  MoveL 631 to (-33.29, -26.54, 35) mm, rotated rx 180 ry 0 rz -180 deg; joints [31.763, 57.392, 24.529, -147.981, 83.138, -184.273]
  Call Extruder(6882.338)
  MoveL 632 to (-26.54, -33.28, 35) mm, rotated rx 180 ry 0 rz -180 deg; joints [30.206, 57.574, 23.981, -149.522, 82.708, -184.272]
  Call Extruder(6897.234)
  MoveL 633 to (-18.47, -38.36, 35) mm, rotated rx 180 ry 0 rz 180 deg; joints [28.808, 57.937, 22.898, -150.881, 81.977, -184.445]
  Call Extruder(6912.129)
  MoveL 634 to (-9.47, -41.5, 35) mm, rotated rx 180 ry 0 rz 180 deg; joints [27.654, 58.472, 21.339, -151.97, 80.985, -184.769]
  Call Extruder(6927.025)
  MoveL 635 to (0, -42.57, 35) mm, rotated rx 180 ry 0 rz 180 deg; joints [26.805, 59.159, 19.387, -152.729, 79.791, -185.221]
  Call Extruder(6928.241)
  MoveL 636 to (0.77, -42.49, 35) mm, rotated rx -180 ry 0 rz 180 deg; joints [26.762, 59.224, 19.206, -152.762, 79.683, -185.267]
  Call Extruder(6941.921)
  MoveL 637 to (9.47, -41.5, 35) mm, rotated rx 180 ry 0 rz -180 deg; joints [26.29, 59.972, 17.142, -153.125, 78.466, -185.786]
  Call Extruder(6956.817)
  MoveL 638 to (18.47, -38.36, 35) mm, rotated rx -180 ry 0 rz -180 deg; joints [26.114, 60.875, 14.715, -153.155, 77.088, -186.452]
  Call Extruder(6971.713)
  MoveL 639 to (26.54, -33.28, 35) mm, rotated rx -180 ry 0 rz -180 deg; joints [26.262, 61.827, 12.225, -152.835, 75.735, -187.206]
  Call Extruder(6986.609)
  MoveL 640 to (33.28, -26.54, 35) mm, rotated rx 180 ry 0 rz 180 deg; joints [26.703, 62.779, 9.793, -152.201, 74.481, -188.03]
  Call Extruder(7001.504)
  MoveL 641 to (38.36, -18.47, 35) mm, rotated rx 180 ry 0 rz -180 deg; joints [27.4, 63.681, 7.536, -151.299, 73.389, -188.896]
  Call Extruder(7016.400)
  MoveL 642 to (41.5, -9.47, 35) mm, rotated rx -180 ry 0 rz -180 deg; joints [28.309, 64.481, 5.567, -150.186, 72.517, -189.768]
  Call Extruder(7031.296)
  MoveL 643 to (42.57, 0, 35) mm, rotated rx -180 ry 0 rz 180 deg; joints [29.382, 65.132, 3.985, -148.925, 71.904, -190.602]
  Call Extruder(7046.192)
  MoveL 644 to (41.51, 9.47, 35) mm, rotated rx -180 ry 0 rz -180 deg; joints [30.575, 65.593, 2.875, -147.579, 71.579, -191.348]
  Call Extruder(7061.087)
  MoveL 645 to (38.36, 18.47, 35) mm, rotated rx -180 ry 0 rz -180 deg; joints [31.839, 65.836, 2.295, -146.213, 71.552, -191.955]
  Call Extruder(7075.983)
  MoveL 646 to (33.28, 26.54, 35) mm, rotated rx 180 ry 0 rz -180 deg; joints [33.128, 65.843, 2.278, -144.884, 71.816, -192.378]
  Call Extruder(7090.879)
  MoveL 647 to (26.54, 33.29, 35) mm, rotated rx 180 ry 0 rz -180 deg; joints [34.394, 65.614, 2.825, -143.644, 72.348, -192.583]
  Call Extruder(7105.775)
  MoveL 648 to (18.47, 38.36, 35) mm, rotated rx 180 ry 0 rz -180 deg; joints [35.592, 65.165, 3.906, -142.537, 73.113, -192.549]
  Call Extruder(7120.671)
  MoveL 649 to (9.47, 41.5, 35) mm, rotated rx 180 ry 0 rz 180 deg; joints [36.675, 64.524, 5.462, -141.601, 74.068, -192.274]
  Call Extruder(7135.566)
  MoveL 650 to (0, 42.57, 35) mm, rotated rx 180 ry 0 rz 180 deg; joints [37.594, 63.731, 7.411, -140.868, 75.161, -191.77]
  Call Extruder(7150.462)
  MoveL 651 to (-9.47, 41.5, 35) mm, rotated rx 180 ry 0 rz 180 deg; joints [38.304, 62.834, 9.654, -140.366, 76.342, -191.066]
  Call Extruder(7165.358)
  MoveL 652 to (-18.47, 38.36, 35) mm, rotated rx 180 ry 0 rz -180 deg; joints [38.762, 61.883, 12.079, -140.123, 77.56, -190.202]
  Call Extruder(7180.254)
  MoveL 653 to (-26.54, 33.29, 35) mm, rotated rx 180 ry 0 rz -180 deg; joints [38.928, 60.93, 14.569, -140.162, 78.768, -189.23]
  Call Extruder(7195.150)
  MoveL 654 to (-33.29, 26.54, 35) mm, rotated rx -180 ry 0 rz 180 deg; joints [38.772, 60.023, 17.003, -140.502, 79.919, -188.21]
  Call Extruder(7210.046)
  MoveL 655 to (-38.36, 18.47, 35) mm, rotated rx -180 ry 0 rz 180 deg; joints [38.277, 59.204, 19.262, -141.153, 80.969, -187.205]
  Call Extruder(7224.941)
  MoveL 656 to (-41.51, 9.47, 35) mm, rotated rx 180 ry 0 rz 180 deg; joints [37.447, 58.508, 21.234, -142.107, 81.872, -186.279]
  Call Extruder(7239.837)
  MoveL 657 to (-42.57, 0, 35) mm, rotated rx 180 ry 0 rz -180 deg; joints [36.31, 57.964, 22.819, -143.334, 82.584, -185.489]
  Call Extruder(7247.391)
  MoveL 658 to (-42.03, -4.8, 35) mm, rotated rx 180 ry 0 rz 180 deg; joints [35.612, 57.771, 23.391, -144.064, 82.824, -185.174]
  Set speed (130.0 mm/s)
  MoveL 659 to (-54.1, -7.67, 35) mm, rotated rx 180 ry 0 rz -180 deg; joints [36.421, 56.883, 26.099, -143.373, 84.357, -184.181]
  Call Extruder(7251.464)
  Set speed (30.0 mm/s)
  MoveL 660 to (-53.59, -12.23, 35) mm, rotated rx 180 ry 0 rz -180 deg; joints [35.732, 56.714, 26.627, -144.084, 84.599, -183.9]
  Call Extruder(7262.394)
  MoveL 661 to (-49.53, -23.85, 35) mm, rotated rx 180 ry 0 rz -180 deg; joints [33.663, 56.476, 27.386, -146.185, 84.894, -183.411]
  Call Extruder(7273.324)
  MoveL 662 to (-42.98, -34.27, 35) mm, rotated rx -180 ry 0 rz 180 deg; joints [31.506, 56.469, 27.408, -148.348, 84.782, -183.209]
  Call Extruder(7284.255)
  MoveL 663 to (-34.27, -42.98, 35) mm, rotated rx 180 ry 0 rz 180 deg; joints [29.427, 56.694, 26.692, -150.409, 84.242, -183.261]
  Call Extruder(7295.185)
  MoveL 664 to (-23.85, -49.52, 35) mm, rotated rx 180 ry 0 rz 180 deg; joints [27.581, 57.146, 25.28, -152.213, 83.292, -183.522]
  Call Extruder(7306.115)
  MoveL 665 to (-12.23, -53.59, 35) mm, rotated rx 180 ry 0 rz 180 deg; joints [26.087, 57.817, 23.254, -153.636, 81.987, -183.952]
  Call Extruder(7317.045)
  MoveL 666 to (0, -54.97, 35) mm, rotated rx 180 ry 0 rz -180 deg; joints [25.019, 58.686, 20.723, -154.602, 80.413, -184.521]
  Call Extruder(7318.968)
  MoveL 667 to (2.15, -54.73, 35) mm, rotated rx 180 ry 0 rz -180 deg; joints [24.908, 58.864, 20.219, -154.69, 80.109, -184.644]
  Call Extruder(7327.975)
  MoveL 668 to (12.23, -53.59, 35) mm, rotated rx 180 ry 0 rz 180 deg; joints [24.406, 59.724, 17.819, -155.077, 78.672, -185.215]
  Call Extruder(7338.905)
  MoveL 669 to (23.85, -49.53, 35) mm, rotated rx -180 ry 0 rz 180 deg; joints [24.239, 60.887, 14.685, -155.066, 76.867, -186.03]
  Call Extruder(7349.836)
  MoveL 670 to (34.27, -42.98, 35) mm, rotated rx 180 ry 0 rz 180 deg; joints [24.487, 62.12, 11.47, -154.602, 75.102, -186.96]
  Call Extruder(7360.766)
  MoveL 671 to (42.98, -34.27, 35) mm, rotated rx 180 ry 0 rz 180 deg; joints [25.101, 63.363, 8.326, -153.736, 73.471, -187.991]
  Call Extruder(7371.696)
  MoveL 672 to (49.52, -23.85, 35) mm, rotated rx 180 ry 0 rz 180 deg; joints [26.025, 64.548, 5.404, -152.536, 72.058, -189.097]
  Call Extruder(7382.626)
  MoveL 673 to (53.59, -12.23, 35) mm, rotated rx -180 ry 0 rz -180 deg; joints [27.2, 65.605, 2.847, -151.077, 70.933, -190.232]
  Call Extruder(7393.557)
  MoveL 674 to (54.97, 0, 35) mm, rotated rx 180 ry 0 rz -180 deg; joints [28.57, 66.47, 0.786, -149.44, 70.152, -191.336]
  Call Extruder(7404.487)
  MoveL 675 to (53.59, 12.23, 35) mm, rotated rx 180 ry 0 rz 180 deg; joints [30.077, 67.087, -0.665, -147.712, 69.749, -192.338]
  Call Extruder(7415.417)
  MoveL 676 to (49.52, 23.85, 35) mm, rotated rx -180 ry 0 rz -180 deg; joints [31.665, 67.411, -1.424, -145.972, 69.735, -193.163]
  Call Extruder(7426.347)
  MoveL 677 to (42.98, 34.27, 35) mm, rotated rx 180 ry 0 rz -180 deg; joints [33.282, 67.42, -1.445, -144.295, 70.101, -193.745]
  Call Extruder(7437.277)
  MoveL 678 to (34.27, 42.98, 35) mm, rotated rx 180 ry 0 rz -180 deg; joints [34.874, 67.114, -0.729, -142.742, 70.813, -194.035]
  Call Extruder(7448.208)
  MoveL 679 to (23.85, 49.53, 35) mm, rotated rx 180 ry 0 rz -180 deg; joints [36.387, 66.514, 0.683, -141.362, 71.82, -194.004]
  Call Extruder(7459.138)
  MoveL 680 to (12.23, 53.59, 35) mm, rotated rx -180 ry 0 rz -180 deg; joints [37.766, 65.662, 2.71, -140.192, 73.06, -193.649]
  Call Extruder(7470.068)
  MoveL 681 to (0, 54.97, 35) mm, rotated rx -180 ry 0 rz -180 deg; joints [38.954, 64.614, 5.242, -139.267, 74.466, -192.987]
  Call Extruder(7480.998)
  MoveL 682 to (-12.23, 53.59, 35) mm, rotated rx 180 ry 0 rz -180 deg; joints [39.895, 63.435, 8.147, -138.616, 75.972, -192.056]
  Call Extruder(7491.928)
  MoveL 683 to (-23.85, 49.52, 35) mm, rotated rx -180 ry 0 rz 180 deg; joints [40.528, 62.194, 11.282, -138.274, 77.515, -190.912]
  Call Extruder(7502.859)
  MoveL 684 to (-34.27, 42.98, 35) mm, rotated rx 180 ry 0 rz 180 deg; joints [40.799, 60.958, 14.496, -138.275, 79.04, -189.622]
  Call Extruder(7513.789)
  MoveL 685 to (-42.98, 34.27, 35) mm, rotated rx 180 ry 0 rz 180 deg; joints [40.659, 59.789, 17.64, -138.653, 80.496, -188.267]
  Call Extruder(7524.719)
  MoveL 686 to (-49.53, 23.85, 35) mm, rotated rx -180 ry 0 rz -180 deg; joints [40.072, 58.743, 20.561, -139.432, 81.835, -186.932]
  Call Extruder(7535.649)
  MoveL 687 to (-53.59, 12.23, 35) mm, rotated rx 180 ry 0 rz 180 deg; joints [39.031, 57.863, 23.118, -140.62, 83.005, -185.708]
  Call Extruder(7546.579)
  MoveL 688 to (-54.97, 0, 35) mm, rotated rx 180 ry 0 rz 180 deg; joints [37.56, 57.18, 25.177, -142.193, 83.948, -184.676]
  Call Extruder(7552.105)
  MoveL 689 to (-54.27, -6.18, 35) mm, rotated rx 180 ry 0 rz -180 deg; joints [36.644, 56.939, 25.923, -143.142, 84.278, -184.275]
  Set speed (130.0 mm/s)
  MoveL 690 to (-49.9, -9.51, 35) mm, rotated rx 180 ry 0 rz 180 deg; joints [35.741, 57.057, 25.556, -144.032, 84.01, -184.331]
  MoveL 691 to (2.97, -12.99, 35) mm, rotated rx 180 ry 0 rz 180 deg; joints [30.614, 60.72, 15.128, -148.606, 77.853, -187.317]
  Call Extruder(7556.769)
  Set speed (80.0 mm/s)
  MoveL 692 to (5.78, -12.01, 35) mm, rotated rx 180 ry 0 rz 180 deg; joints [30.526, 61.006, 14.369, -148.642, 77.438, -187.55]
  Call Extruder(7561.432)
  MoveL 693 to (8.31, -10.42, 35) mm, rotated rx -180 ry 0 rz 180 deg; joints [30.538, 61.302, 13.59, -148.572, 77.027, -187.811]
  Call Extruder(7566.096)
  MoveL 694 to (10.42, -8.31, 35) mm, rotated rx 180 ry 0 rz 180 deg; joints [30.649, 61.594, 12.829, -148.402, 76.643, -188.088]
  Call Extruder(7570.760)
  MoveL 695 to (12.01, -5.78, 35) mm, rotated rx 180 ry 0 rz 180 deg; joints [30.85, 61.866, 12.124, -148.143, 76.304, -188.37]
  Call Extruder(7575.424)
  MoveL 696 to (12.99, -2.97, 35) mm, rotated rx 180 ry 0 rz -180 deg; joints [31.131, 62.104, 11.511, -147.808, 76.027, -188.643]
  Call Extruder(7580.087)
  MoveL 697 to (13.33, 0, 35) mm, rotated rx -180 ry 0 rz 180 deg; joints [31.476, 62.296, 11.021, -147.416, 75.828, -188.894]
  Call Extruder(7584.751)
  MoveL 698 to (12.99, 2.97, 35) mm, rotated rx -180 ry 0 rz -180 deg; joints [31.869, 62.43, 10.678, -146.987, 75.714, -189.109]
  Call Extruder(7589.415)
  MoveL 699 to (12.01, 5.78, 35) mm, rotated rx 180 ry 0 rz -180 deg; joints [32.292, 62.5, 10.5, -146.541, 75.691, -189.276]
  Call Extruder(7594.079)
  MoveL 700 to (10.42, 8.31, 35) mm, rotated rx 180 ry 0 rz 180 deg; joints [32.725, 62.502, 10.494, -146.1, 75.758, -189.387]
  Call Extruder(7598.743)
  MoveL 701 to (8.31, 10.42, 35) mm, rotated rx 180 ry 0 rz 180 deg; joints [33.149, 62.436, 10.663, -145.683, 75.912, -189.433]
  Call Extruder(7603.406)
  MoveL 702 to (5.78, 12.01, 35) mm, rotated rx 180 ry 0 rz -180 deg; joints [33.544, 62.305, 10.997, -145.309, 76.144, -189.412]
  Call Extruder(7608.070)
  MoveL 703 to (2.97, 13, 35) mm, rotated rx 180 ry 0 rz 180 deg; joints [33.893, 62.117, 11.479, -144.996, 76.442, -189.323]
  Call Extruder(7612.734)
  MoveL 704 to (0, 13.33, 35) mm, rotated rx 180 ry 0 rz 180 deg; joints [34.177, 61.881, 12.085, -144.758, 76.791, -189.171]
  Call Extruder(7617.398)
  MoveL 705 to (-2.97, 13, 35) mm, rotated rx 180 ry 0 rz -180 deg; joints [34.384, 61.611, 12.785, -144.607, 77.174, -188.963]
  Call Extruder(7622.062)
  MoveL 706 to (-5.78, 12.01, 35) mm, rotated rx 180 ry 0 rz -180 deg; joints [34.5, 61.32, 13.544, -144.55, 77.573, -188.711]
  Call Extruder(7626.725)
  MoveL 707 to (-8.31, 10.42, 35) mm, rotated rx -180 ry 0 rz 180 deg; joints [34.518, 61.023, 14.324, -144.592, 77.97, -188.428]
  Call Extruder(7631.389)
  MoveL 708 to (-10.42, 8.31, 35) mm, rotated rx 180 ry 0 rz 180 deg; joints [34.436, 60.736, 15.085, -144.733, 78.344, -188.131]
  Call Extruder(7636.053)
  MoveL 709 to (-12.01, 5.78, 35) mm, rotated rx 180 ry 0 rz -180 deg; joints [34.254, 60.472, 15.79, -144.968, 78.68, -187.835]
  Call Extruder(7640.717)
  MoveL 710 to (-13, 2.97, 35) mm, rotated rx -180 ry 0 rz -180 deg; joints [33.981, 60.244, 16.404, -145.287, 78.96, -187.557]
  Call Extruder(7645.380)
  MoveL 711 to (-13.33, 0, 35) mm, rotated rx 180 ry 0 rz -180 deg; joints [33.63, 60.063, 16.894, -145.676, 79.169, -187.311]
  Call Extruder(7650.044)
  MoveL 712 to (-13, -2.97, 35) mm, rotated rx 180 ry 0 rz 180 deg; joints [33.218, 59.936, 17.238, -146.116, 79.297, -187.109]
  Call Extruder(7654.708)
  MoveL 713 to (-12.01, -5.78, 35) mm, rotated rx 180 ry 0 rz -180 deg; joints [32.767, 59.871, 17.417, -146.583, 79.337, -186.961]
  Call Extruder(7659.372)
  MoveL 714 to (-10.42, -8.31, 35) mm, rotated rx 180 ry 0 rz -180 deg; joints [32.302, 59.869, 17.422, -147.052, 79.283, -186.872]
  Call Extruder(7664.036)
  MoveL 715 to (-8.31, -10.42, 35) mm, rotated rx 180 ry 0 rz 180 deg; joints [31.85, 59.931, 17.253, -147.498, 79.139, -186.845]
  Call Extruder(7668.699)
  MoveL 716 to (-5.78, -12.01, 35) mm, rotated rx -180 ry 0 rz -180 deg; joints [31.435, 60.054, 16.919, -147.896, 78.911, -186.881]
  Call Extruder(7673.363)
  MoveL 717 to (-2.97, -12.99, 35) mm, rotated rx 180 ry 0 rz -180 deg; joints [31.079, 60.232, 16.436, -148.224, 78.61, -186.975]
  Call Extruder(7678.027)
  MoveL 718 to (0, -13.33, 35) mm, rotated rx 180 ry 0 rz 180 deg; joints [30.801, 60.457, 15.829, -148.465, 78.251, -187.123]
  Call Extruder(7682.691)
  MoveL 719 to (2.97, -12.99, 35) mm, rotated rx 180 ry 0 rz 180 deg; joints [30.614, 60.72, 15.128, -148.606, 77.853, -187.317]
  Set speed (130.0 mm/s)
  MoveL 720 to (2.97, -12.99, 40) mm, rotated rx 180 ry 0 rz 180 deg; joints [30.614, 59.777, 15.612, -148.554, 77.462, -187.562]
  MoveL 721 to (-26.25, -4.54, 40) mm, rotated rx 180 ry 0 rz 180 deg; joints [34.172, 57.891, 20.698, -145.294, 80.579, -186.468]
  Call Extruder(7684.924)
  Set speed (60.0 mm/s)
  MoveL 722 to (-26.09, -5.96, 40) mm, rotated rx 180 ry 0 rz -180 deg; joints [33.969, 57.832, 20.861, -145.509, 80.642, -186.374]
  Call Extruder(7694.288)
  MoveL 723 to (-24.12, -11.61, 40) mm, rotated rx -180 ry 0 rz -180 deg; joints [33.033, 57.703, 21.223, -146.473, 80.733, -186.09]
  Call Extruder(7703.653)
  MoveL 724 to (-20.93, -16.69, 40) mm, rotated rx 180 ry 0 rz 180 deg; joints [32.066, 57.699, 21.234, -147.448, 80.638, -185.928]
  Call Extruder(7713.018)
  MoveL 725 to (-16.69, -20.93, 40) mm, rotated rx 180 ry 0 rz -180 deg; joints [31.126, 57.821, 20.892, -148.376, 80.355, -185.89]
  Call Extruder(7722.383)
  MoveL 726 to (-11.61, -24.11, 40) mm, rotated rx 180 ry 0 rz -180 deg; joints [30.272, 58.064, 20.217, -149.2, 79.897, -185.97]
  Call Extruder(7731.748)
  MoveL 727 to (-5.96, -26.09, 40) mm, rotated rx 180 ry 0 rz -180 deg; joints [29.552, 58.419, 19.242, -149.87, 79.287, -186.158]
  Call Extruder(7741.113)
  MoveL 728 to (0, -26.77, 40) mm, rotated rx 180 ry 0 rz 180 deg; joints [29.003, 58.87, 18.019, -150.351, 78.558, -186.443]
  Call Extruder(7745.379)
  MoveL 729 to (2.71, -26.46, 40) mm, rotated rx -180 ry 0 rz 180 deg; joints [28.841, 59.109, 17.38, -150.474, 78.191, -186.612]
  Call Extruder(7750.478)
  MoveL 730 to (5.96, -26.09, 40) mm, rotated rx -180 ry 0 rz -180 deg; joints [28.65, 59.398, 16.61, -150.618, 77.75, -186.813]
  Call Extruder(7759.843)
  MoveL 731 to (11.61, -24.11, 40) mm, rotated rx -180 ry 0 rz -180 deg; joints [28.503, 59.979, 15.084, -150.664, 76.908, -187.255]
  Call Extruder(7769.208)
  MoveL 732 to (16.69, -20.93, 40) mm, rotated rx 180 ry 0 rz 180 deg; joints [28.559, 60.584, 13.519, -150.493, 76.079, -187.754]
  Call Extruder(7778.573)
  MoveL 733 to (20.93, -16.69, 40) mm, rotated rx 180 ry 0 rz -180 deg; joints [28.808, 61.183, 11.99, -150.121, 75.307, -188.291]
  Call Extruder(7787.938)
  MoveL 734 to (24.12, -11.61, 40) mm, rotated rx -180 ry 0 rz 180 deg; joints [29.229, 61.746, 10.575, -149.575, 74.632, -188.846]
  Call Extruder(7797.303)
  MoveL 735 to (26.09, -5.96, 40) mm, rotated rx -180 ry 0 rz 180 deg; joints [29.796, 62.241, 9.343, -148.888, 74.089, -189.395]
  Call Extruder(7806.668)
  MoveL 736 to (26.77, 0, 40) mm, rotated rx 180 ry 0 rz 180 deg; joints [30.482, 62.641, 8.356, -148.096, 73.703, -189.909]
  Call Extruder(7816.033)
  MoveL 737 to (26.09, 5.96, 40) mm, rotated rx 180 ry 0 rz -180 deg; joints [31.252, 62.923, 7.666, -147.241, 73.493, -190.36]
  Call Extruder(7825.398)
  MoveL 738 to (24.11, 11.61, 40) mm, rotated rx -180 ry 0 rz -180 deg; joints [32.076, 63.07, 7.305, -146.362, 73.466, -190.722]
  Call Extruder(7834.763)
  MoveL 739 to (20.93, 16.69, 40) mm, rotated rx -180 ry 0 rz 180 deg; joints [32.917, 63.074, 7.295, -145.499, 73.619, -190.97]
  Call Extruder(7844.128)
  MoveL 740 to (16.69, 20.93, 40) mm, rotated rx 180 ry 0 rz 180 deg; joints [33.742, 62.935, 7.635, -144.689, 73.942, -191.086]
  Call Extruder(7853.493)
  MoveL 741 to (11.61, 24.12, 40) mm, rotated rx 180 ry 0 rz -180 deg; joints [34.517, 62.661, 8.307, -143.964, 74.414, -191.06]
  Call Extruder(7862.858)
  MoveL 742 to (5.96, 26.09, 40) mm, rotated rx 180 ry 0 rz 180 deg; joints [35.208, 62.267, 9.278, -143.354, 75.01, -190.891]
  Call Extruder(7872.223)
  MoveL 743 to (0, 26.77, 40) mm, rotated rx 180 ry 0 rz -180 deg; joints [35.784, 61.777, 10.497, -142.884, 75.701, -190.587]
  Call Extruder(7881.588)
  MoveL 744 to (-5.96, 26.09, 40) mm, rotated rx 180 ry 0 rz -180 deg; joints [36.214, 61.218, 11.903, -142.576, 76.452, -190.163]
  Call Extruder(7890.953)
  MoveL 745 to (-11.61, 24.12, 40) mm, rotated rx 180 ry 0 rz 180 deg; joints [36.473, 60.62, 13.427, -142.445, 77.231, -189.644]
  Call Extruder(7900.318)
  MoveL 746 to (-16.69, 20.93, 40) mm, rotated rx 180 ry 0 rz 180 deg; joints [36.542, 60.014, 14.993, -142.504, 78.004, -189.06]
  Call Extruder(7909.683)
  MoveL 747 to (-20.93, 16.69, 40) mm, rotated rx 180 ry 0 rz -180 deg; joints [36.407, 59.431, 16.522, -142.759, 78.736, -188.446]
  Call Extruder(7919.048)
  MoveL 748 to (-24.12, 11.61, 40) mm, rotated rx -180 ry 0 rz -180 deg; joints [36.065, 58.899, 17.941, -143.206, 79.395, -187.837]
  Call Extruder(7928.413)
  MoveL 749 to (-26.09, 5.96, 40) mm, rotated rx -180 ry 0 rz 180 deg; joints [35.528, 58.443, 19.177, -143.832, 79.951, -187.269]
  Call Extruder(7937.778)
  MoveL 750 to (-26.77, 0, 40) mm, rotated rx -180 ry 0 rz -180 deg; joints [34.817, 58.082, 20.167, -144.612, 80.375, -186.773]
  Call Extruder(7942.567)
  MoveL 751 to (-26.42, -3.05, 40) mm, rotated rx 180 ry 0 rz -180 deg; joints [34.385, 57.953, 20.525, -145.069, 80.512, -186.567]
  Set speed (130.0 mm/s)
  MoveL 752 to (-41.86, -6.29, 40) mm, rotated rx 180 ry 0 rz 180 deg; joints [35.393, 56.711, 24.057, -144.253, 82.485, -185.378]
  Call Extruder(7947.564)
  Set speed (60.0 mm/s)
  MoveL 753 to (-41.51, -9.47, 40) mm, rotated rx 180 ry 0 rz 180 deg; joints [34.924, 56.586, 24.424, -144.743, 82.639, -185.175]
  Call Extruder(7962.460)
  MoveL 754 to (-38.36, -18.47, 40) mm, rotated rx 180 ry 0 rz 180 deg; joints [33.373, 56.389, 25.006, -146.328, 82.822, -184.759]
  Call Extruder(7977.356)
  MoveL 755 to (-33.29, -26.54, 40) mm, rotated rx 180 ry 0 rz 180 deg; joints [31.763, 56.383, 25.023, -147.947, 82.701, -184.549]
  Call Extruder(7992.252)
  MoveL 756 to (-26.54, -33.28, 40) mm, rotated rx 180 ry 0 rz 180 deg; joints [30.206, 56.569, 24.474, -149.487, 82.267, -184.534]
  Call Extruder(8007.148)
  MoveL 757 to (-18.47, -38.36, 40) mm, rotated rx 180 ry 0 rz 180 deg; joints [28.808, 56.941, 23.389, -150.845, 81.536, -184.694]
  Call Extruder(8022.043)
  MoveL 758 to (-9.47, -41.51, 40) mm, rotated rx 180 ry 0 rz 180 deg; joints [27.654, 57.488, 21.827, -151.932, 80.548, -185.005]
  Call Extruder(8036.939)
  MoveL 759 to (0, -42.57, 40) mm, rotated rx 180 ry 0 rz 180 deg; joints [26.805, 58.189, 19.873, -152.688, 79.361, -185.446]
  Call Extruder(8043.970)
  MoveL 760 to (4.47, -42.07, 40) mm, rotated rx 180 ry 0 rz 180 deg; joints [26.559, 58.574, 18.819, -152.878, 78.742, -185.71]
  Call Extruder(8051.835)
  MoveL 761 to (9.47, -41.5, 40) mm, rotated rx 180 ry 0 rz -180 deg; joints [26.29, 59.017, 17.626, -153.081, 78.046, -186.004]
  Call Extruder(8066.731)
  MoveL 762 to (18.47, -38.36, 40) mm, rotated rx 180 ry 0 rz 180 deg; joints [26.114, 59.935, 15.198, -153.107, 76.681, -186.664]
  Call Extruder(8081.626)
  MoveL 763 to (26.54, -33.28, 40) mm, rotated rx 180 ry 0 rz 180 deg; joints [26.262, 60.901, 12.708, -152.783, 75.341, -187.415]
  Call Extruder(8096.522)
  MoveL 764 to (33.28, -26.54, 40) mm, rotated rx 180 ry 0 rz 180 deg; joints [26.703, 61.865, 10.277, -152.144, 74.1, -188.238]
  Call Extruder(8111.418)
  MoveL 765 to (38.36, -18.47, 40) mm, rotated rx 180 ry 0 rz 180 deg; joints [27.4, 62.777, 8.021, -151.238, 73.023, -189.105]
  Call Extruder(8126.314)
  MoveL 766 to (41.51, -9.47, 40) mm, rotated rx -180 ry 0 rz 180 deg; joints [28.309, 63.586, 6.054, -150.121, 72.163, -189.981]
  Call Extruder(8141.210)
  MoveL 767 to (42.57, 0, 40) mm, rotated rx 180 ry 0 rz 180 deg; joints [29.382, 64.243, 4.474, -148.856, 71.562, -190.82]
  Call Extruder(8156.106)
  MoveL 768 to (41.5, 9.47, 40) mm, rotated rx 180 ry 0 rz 180 deg; joints [30.575, 64.709, 3.365, -147.508, 71.247, -191.571]
  Call Extruder(8171.001)
  MoveL 769 to (38.36, 18.47, 40) mm, rotated rx -180 ry 0 rz 180 deg; joints [31.839, 64.953, 2.786, -146.139, 71.227, -192.185]
  Call Extruder(8185.897)
  MoveL 770 to (33.28, 26.54, 40) mm, rotated rx 180 ry 0 rz -180 deg; joints [33.128, 64.96, 2.77, -144.809, 71.496, -192.615]
  Call Extruder(8200.793)
  MoveL 771 to (26.54, 33.29, 40) mm, rotated rx 180 ry 0 rz -180 deg; joints [34.394, 64.729, 3.316, -143.569, 72.031, -192.828]
  Call Extruder(8215.689)
  MoveL 772 to (18.47, 38.36, 40) mm, rotated rx 180 ry 0 rz -180 deg; joints [35.592, 64.276, 4.395, -142.463, 72.796, -192.803]
  Call Extruder(8230.584)
  MoveL 773 to (9.47, 41.51, 40) mm, rotated rx 180 ry 0 rz 180 deg; joints [36.675, 63.629, 5.949, -141.528, 73.749, -192.537]
  Call Extruder(8245.480)
  MoveL 774 to (0, 42.57, 40) mm, rotated rx -180 ry 0 rz 180 deg; joints [37.594, 62.828, 7.896, -140.797, 74.837, -192.043]
  Call Extruder(8260.376)
  MoveL 775 to (-9.47, 41.51, 40) mm, rotated rx 180 ry 0 rz -180 deg; joints [38.304, 61.921, 10.138, -140.299, 76.012, -191.348]
  Call Extruder(8275.272)
  MoveL 776 to (-18.47, 38.36, 40) mm, rotated rx 180 ry 0 rz -180 deg; joints [38.762, 60.958, 12.563, -140.059, 77.221, -190.493]
  Call Extruder(8290.168)
  MoveL 777 to (-26.54, 33.29, 40) mm, rotated rx 180 ry 0 rz 180 deg; joints [38.928, 59.991, 15.053, -140.103, 78.418, -189.528]
  Call Extruder(8305.063)
  MoveL 778 to (-33.29, 26.54, 40) mm, rotated rx -180 ry 0 rz 180 deg; joints [38.772, 59.069, 17.487, -140.448, 79.557, -188.514]
  Call Extruder(8319.959)
  MoveL 779 to (-38.36, 18.47, 40) mm, rotated rx 180 ry 0 rz 180 deg; joints [38.277, 58.234, 19.748, -141.104, 80.593, -187.512]
  Call Extruder(8334.855)
  MoveL 780 to (-41.5, 9.47, 40) mm, rotated rx 180 ry 0 rz -180 deg; joints [37.447, 57.525, 21.723, -142.062, 81.482, -186.586]
  Call Extruder(8349.751)
  MoveL 781 to (-42.57, 0, 40) mm, rotated rx 180 ry 0 rz 180 deg; joints [36.31, 56.969, 23.309, -143.294, 82.179, -185.793]
  Call Extruder(8357.305)
  MoveL 782 to (-42.03, -4.8, 40) mm, rotated rx 180 ry 0 rz -180 deg; joints [35.612, 56.771, 23.882, -144.025, 82.413, -185.475]
  Set speed (130.0 mm/s)
  MoveL 783 to (-54.1, -7.67, 40) mm, rotated rx -180 ry 0 rz -180 deg; joints [36.421, 55.86, 26.595, -143.341, 83.935, -184.496]
  Call Extruder(8361.378)
  Set speed (30.0 mm/s)
  MoveL 784 to (-53.59, -12.23, 40) mm, rotated rx 180 ry 0 rz 180 deg; joints [35.732, 55.687, 27.125, -144.054, 84.171, -184.212]
  Call Extruder(8372.308)
  MoveL 785 to (-49.53, -23.85, 40) mm, rotated rx 180 ry 0 rz 180 deg; joints [33.663, 55.442, 27.885, -146.157, 84.45, -183.71]
  Call Extruder(8383.238)
  MoveL 786 to (-42.98, -34.27, 40) mm, rotated rx 180 ry 0 rz 180 deg; joints [31.506, 55.435, 27.907, -148.321, 84.327, -183.491]
  Call Extruder(8394.168)
  MoveL 787 to (-34.27, -42.98, 40) mm, rotated rx 180 ry 0 rz 180 deg; joints [29.427, 55.666, 27.189, -150.382, 83.781, -183.524]
  Call Extruder(8405.099)
  MoveL 788 to (-23.85, -49.52, 40) mm, rotated rx 180 ry 0 rz -180 deg; joints [27.581, 56.131, 25.775, -152.183, 82.831, -183.767]
  Call Extruder(8416.029)
  MoveL 789 to (-12.23, -53.59, 40) mm, rotated rx 180 ry 0 rz 180 deg; joints [26.087, 56.818, 23.745, -153.604, 81.532, -184.18]
  Call Extruder(8426.959)
  MoveL 790 to (0, -54.97, 40) mm, rotated rx 180 ry 0 rz 180 deg; joints [25.019, 57.707, 21.211, -154.565, 79.969, -184.735]
  Call Extruder(8432.187)
  MoveL 791 to (5.85, -54.31, 40) mm, rotated rx 180 ry 0 rz 180 deg; joints [24.72, 58.204, 19.831, -154.798, 79.146, -185.064]
  Call Extruder(8437.889)
  MoveL 792 to (12.23, -53.59, 40) mm, rotated rx -180 ry 0 rz 180 deg; joints [24.406, 58.765, 18.304, -155.036, 78.242, -185.42]
  Call Extruder(8448.819)
  MoveL 793 to (23.85, -49.52, 40) mm, rotated rx 180 ry 0 rz 180 deg; joints [24.239, 59.947, 15.168, -155.02, 76.454, -186.228]
  Call Extruder(8459.750)
  MoveL 794 to (34.27, -42.98, 40) mm, rotated rx 180 ry 0 rz -180 deg; joints [24.487, 61.198, 11.953, -154.551, 74.706, -187.155]
  Call Extruder(8470.680)
  MoveL 795 to (42.98, -34.27, 40) mm, rotated rx -180 ry 0 rz -180 deg; joints [25.101, 62.456, 8.811, -153.68, 73.093, -188.186]
  Call Extruder(8481.610)
  MoveL 796 to (49.52, -23.85, 40) mm, rotated rx 180 ry 0 rz 180 deg; joints [26.025, 63.653, 5.891, -152.475, 71.697, -189.295]
  Call Extruder(8492.540)
  MoveL 797 to (53.59, -12.23, 40) mm, rotated rx 180 ry 0 rz -180 deg; joints [27.2, 64.72, 3.337, -151.01, 70.589, -190.434]
  Call Extruder(8503.470)
  MoveL 798 to (54.97, 0, 40) mm, rotated rx 180 ry 0 rz 180 deg; joints [28.57, 65.593, 1.28, -149.369, 69.822, -191.544]
  Call Extruder(8514.401)
  MoveL 799 to (53.59, 12.23, 40) mm, rotated rx -180 ry 0 rz -180 deg; joints [30.077, 66.213, -0.168, -147.637, 69.43, -192.552]
  Call Extruder(8525.331)
  MoveL 800 to (49.52, 23.85, 40) mm, rotated rx 180 ry 0 rz 180 deg; joints [31.665, 66.54, -0.925, -145.895, 69.427, -193.386]
  Call Extruder(8536.261)
  MoveL 801 to (42.98, 34.27, 40) mm, rotated rx 180 ry 0 rz 180 deg; joints [33.282, 66.549, -0.947, -144.216, 69.799, -193.977]
  Call Extruder(8547.191)
  MoveL 802 to (34.27, 42.98, 40) mm, rotated rx -180 ry 0 rz 180 deg; joints [34.874, 66.241, -0.232, -142.662, 70.514, -194.277]
  Call Extruder(8558.121)
  MoveL 803 to (23.85, 49.53, 40) mm, rotated rx 180 ry 0 rz 180 deg; joints [36.387, 65.637, 1.177, -141.282, 71.521, -194.257]
  Call Extruder(8569.051)
  MoveL 804 to (12.23, 53.59, 40) mm, rotated rx 180 ry 0 rz -180 deg; joints [37.766, 64.778, 3.201, -140.115, 72.758, -193.912]
  Call Extruder(8579.982)
  MoveL 805 to (0, 54.97, 40) mm, rotated rx 180 ry 0 rz -180 deg; joints [38.954, 63.72, 5.729, -139.192, 74.159, -193.262]
  Call Extruder(8590.912)
  MoveL 806 to (-12.23, 53.59, 40) mm, rotated rx 180 ry 0 rz 180 deg; joints [39.895, 62.529, 8.632, -138.546, 75.656, -192.344]
  Call Extruder(8601.842)
  MoveL 807 to (-23.85, 49.53, 40) mm, rotated rx 180 ry 0 rz -180 deg; joints [40.528, 61.273, 11.765, -138.209, 77.188, -191.211]
  Call Extruder(8612.772)
  MoveL 808 to (-34.27, 42.98, 40) mm, rotated rx 180 ry 0 rz 180 deg; joints [40.799, 60.019, 14.98, -138.216, 78.7, -189.932]
  Call Extruder(8623.702)
  MoveL 809 to (-42.98, 34.27, 40) mm, rotated rx 180 ry 0 rz 180 deg; joints [40.659, 58.831, 18.125, -138.6, 80.141, -188.584]
  Call Extruder(8634.633)
  MoveL 810 to (-49.53, 23.85, 40) mm, rotated rx 180 ry 0 rz 180 deg; joints [40.072, 57.765, 21.049, -139.385, 81.463, -187.255]
  Call Extruder(8645.563)
  MoveL 811 to (-53.59, 12.23, 40) mm, rotated rx 180 ry 0 rz -180 deg; joints [39.031, 56.865, 23.609, -140.58, 82.614, -186.032]
  Call Extruder(8656.493)
  MoveL 812 to (-54.97, 0, 40) mm, rotated rx 180 ry 0 rz 180 deg; joints [37.56, 56.165, 25.672, -142.158, 83.538, -184.997]
  Call Extruder(8662.019)
  MoveL 813 to (-54.27, -6.18, 40) mm, rotated rx -180 ry 0 rz -180 deg; joints [36.644, 55.918, 26.419, -143.109, 83.858, -184.591]
  Set speed (130.0 mm/s)
  MoveL 814 to (-49.9, -9.51, 40) mm, rotated rx 180 ry 0 rz -180 deg; joints [35.741, 56.039, 26.051, -143.999, 83.587, -184.64]
  MoveL 815 to (1.22, -13.19, 40) mm, rotated rx -180 ry 0 rz 180 deg; joints [30.724, 59.619, 16.026, -148.472, 77.694, -187.449]
  Call Extruder(8664.768)
  Set speed (80.0 mm/s)
  MoveL 816 to (2.97, -12.99, 40) mm, rotated rx 180 ry 0 rz 180 deg; joints [30.614, 59.777, 15.612, -148.554, 77.462, -187.562]
  Call Extruder(8669.431)
  MoveL 817 to (5.78, -12.01, 40) mm, rotated rx 180 ry 0 rz -180 deg; joints [30.526, 60.068, 14.853, -148.588, 77.05, -187.793]
  Call Extruder(8674.095)
  MoveL 818 to (8.31, -10.42, 40) mm, rotated rx -180 ry 0 rz 180 deg; joints [30.538, 60.369, 14.073, -148.517, 76.643, -188.052]
  Call Extruder(8678.759)
  MoveL 819 to (10.42, -8.31, 40) mm, rotated rx 180 ry 0 rz -180 deg; joints [30.649, 60.665, 13.312, -148.346, 76.263, -188.329]
  Call Extruder(8683.423)
  MoveL 820 to (12.01, -5.78, 40) mm, rotated rx -180 ry 0 rz -180 deg; joints [30.85, 60.941, 12.607, -148.085, 75.928, -188.611]
  Call Extruder(8688.086)
  MoveL 821 to (12.99, -2.97, 40) mm, rotated rx 180 ry 0 rz -180 deg; joints [31.131, 61.182, 11.995, -147.749, 75.656, -188.885]
  Call Extruder(8692.750)
  MoveL 822 to (13.33, 0, 40) mm, rotated rx -180 ry 0 rz -180 deg; joints [31.476, 61.376, 11.505, -147.356, 75.46, -189.136]
  Call Extruder(8697.414)
  MoveL 823 to (13, 2.97, 40) mm, rotated rx 180 ry 0 rz -180 deg; joints [31.869, 61.512, 11.162, -146.926, 75.35, -189.353]
  Call Extruder(8702.078)
  MoveL 824 to (12.01, 5.78, 40) mm, rotated rx -180 ry 0 rz 180 deg; joints [32.292, 61.583, 10.983, -146.479, 75.329, -189.523]
  Call Extruder(8706.741)
  MoveL 825 to (10.42, 8.31, 40) mm, rotated rx 180 ry 0 rz 180 deg; joints [32.725, 61.585, 10.978, -146.037, 75.399, -189.637]
  Call Extruder(8711.406)
  MoveL 826 to (8.31, 10.42, 40) mm, rotated rx 180 ry 0 rz -180 deg; joints [33.149, 61.518, 11.146, -145.621, 75.554, -189.686]
  Call Extruder(8716.069)
  MoveL 827 to (5.78, 12.01, 40) mm, rotated rx 180 ry 0 rz -180 deg; joints [33.544, 61.385, 11.48, -145.247, 75.786, -189.668]
  Call Extruder(8720.733)
  MoveL 828 to (2.97, 12.99, 40) mm, rotated rx -180 ry 0 rz 180 deg; joints [33.893, 61.195, 11.962, -144.935, 76.083, -189.582]
  Call Extruder(8725.397)
  MoveL 829 to (0, 13.33, 40) mm, rotated rx 180 ry 0 rz -180 deg; joints [34.177, 60.956, 12.569, -144.698, 76.43, -189.433]
  Call Extruder(8730.061)
  MoveL 830 to (-2.97, 12.99, 40) mm, rotated rx 180 ry 0 rz 180 deg; joints [34.384, 60.682, 13.269, -144.547, 76.811, -189.228]
  Call Extruder(8734.724)
  MoveL 831 to (-5.78, 12.01, 40) mm, rotated rx -180 ry 0 rz 180 deg; joints [34.5, 60.386, 14.027, -144.492, 77.207, -188.978]
  Call Extruder(8739.388)
  MoveL 832 to (-8.31, 10.42, 40) mm, rotated rx 180 ry 0 rz -180 deg; joints [34.518, 60.085, 14.807, -144.535, 77.599, -188.698]
  Call Extruder(8744.052)
  MoveL 833 to (-10.42, 8.31, 40) mm, rotated rx 180 ry 0 rz -180 deg; joints [34.436, 59.794, 15.568, -144.677, 77.97, -188.402]
  Call Extruder(8748.716)
  MoveL 834 to (-12.01, 5.78, 40) mm, rotated rx 180 ry 0 rz -180 deg; joints [34.254, 59.525, 16.274, -144.914, 78.301, -188.106]
  Call Extruder(8753.379)
  MoveL 835 to (-12.99, 2.97, 40) mm, rotated rx 180 ry 0 rz -180 deg; joints [33.981, 59.294, 16.888, -145.234, 78.576, -187.828]
  Call Extruder(8758.043)
  MoveL 836 to (-13.33, 0, 40) mm, rotated rx -180 ry 0 rz -180 deg; joints [33.63, 59.109, 17.379, -145.625, 78.782, -187.581]
  Call Extruder(8762.707)
  MoveL 837 to (-13, -2.97, 40) mm, rotated rx 180 ry 0 rz 180 deg; joints [33.218, 58.981, 17.723, -146.065, 78.907, -187.377]
  Call Extruder(8767.371)
  MoveL 838 to (-12.01, -5.78, 40) mm, rotated rx 180 ry 0 rz 180 deg; joints [32.767, 58.914, 17.902, -146.533, 78.943, -187.226]
  Call Extruder(8772.034)
  MoveL 839 to (-10.42, -8.31, 40) mm, rotated rx 180 ry 0 rz -180 deg; joints [32.302, 58.912, 17.907, -147.003, 78.887, -187.134]
  Call Extruder(8776.699)
  MoveL 840 to (-8.31, -10.42, 40) mm, rotated rx 180 ry 0 rz 180 deg; joints [31.85, 58.975, 17.738, -147.449, 78.742, -187.103]
  Call Extruder(8781.362)
  MoveL 841 to (-5.78, -12.01, 40) mm, rotated rx 180 ry 0 rz -180 deg; joints [31.435, 59.1, 17.403, -147.846, 78.514, -187.135]
  Call Extruder(8786.026)
  MoveL 842 to (-2.97, -12.99, 40) mm, rotated rx 180 ry 0 rz 180 deg; joints [31.079, 59.281, 16.92, -148.174, 78.213, -187.226]
  Call Extruder(8790.690)
  MoveL 843 to (0, -13.33, 40) mm, rotated rx 180 ry 0 rz 180 deg; joints [30.801, 59.511, 16.313, -148.414, 77.856, -187.37]
  Call Extruder(8792.605)
  MoveL 844 to (1.22, -13.19, 40) mm, rotated rx -180 ry 0 rz 180 deg; joints [30.724, 59.619, 16.026, -148.472, 77.694, -187.449]
  Set speed (130.0 mm/s)
  MoveL 845 to (1.22, -13.19, 45) mm, rotated rx 180 ry 0 rz -180 deg; joints [30.724, 58.678, 16.493, -148.417, 77.29, -187.704]
  MoveL 846 to (-26.25, -4.54, 45) mm, rotated rx -180 ry 0 rz 180 deg; joints [34.172, 56.918, 21.169, -145.245, 80.166, -186.758]
  Call Extruder(8794.837)
  Set speed (60.0 mm/s)
  MoveL 847 to (-26.09, -5.96, 45) mm, rotated rx 180 ry 0 rz -180 deg; joints [33.969, 56.858, 21.332, -145.461, 80.227, -186.664]
  Call Extruder(8804.202)
  MoveL 848 to (-24.12, -11.61, 45) mm, rotated rx 180 ry 0 rz 180 deg; joints [33.033, 56.726, 21.695, -146.426, 80.312, -186.373]
  Call Extruder(8813.567)
  MoveL 849 to (-20.93, -16.69, 45) mm, rotated rx -180 ry 0 rz 180 deg; joints [32.066, 56.722, 21.705, -147.403, 80.211, -186.205]
  Call Extruder(8822.932)
  MoveL 850 to (-16.69, -20.93, 45) mm, rotated rx 180 ry 0 rz -180 deg; joints [31.126, 56.847, 21.363, -148.331, 79.926, -186.158]
  Call Extruder(8832.297)
  MoveL 851 to (-11.61, -24.11, 45) mm, rotated rx 180 ry 0 rz 180 deg; joints [30.272, 57.095, 20.687, -149.153, 79.468, -186.23]
  Call Extruder(8841.662)
  MoveL 852 to (-5.96, -26.09, 45) mm, rotated rx 180 ry 0 rz 180 deg; joints [29.552, 57.456, 19.711, -149.822, 78.86, -186.41]
  Call Extruder(8851.027)
  MoveL 853 to (0, -26.77, 45) mm, rotated rx -180 ry 0 rz -180 deg; joints [29.003, 57.916, 18.487, -150.301, 78.135, -186.688]
  Call Extruder(8860.392)
  MoveL 854 to (5.96, -26.09, 45) mm, rotated rx 180 ry 0 rz 180 deg; joints [28.65, 58.453, 17.077, -150.566, 77.333, -187.053]
  Call Extruder(8869.757)
  MoveL 855 to (11.61, -24.11, 45) mm, rotated rx 180 ry 0 rz -180 deg; joints [28.503, 59.043, 15.551, -150.609, 76.499, -187.491]
  Call Extruder(8879.122)
  MoveL 856 to (16.69, -20.93, 45) mm, rotated rx -180 ry 0 rz -180 deg; joints [28.559, 59.658, 13.985, -150.436, 75.678, -187.988]
  Call Extruder(8888.487)
  MoveL 857 to (20.93, -16.69, 45) mm, rotated rx 180 ry 0 rz 180 deg; joints [28.808, 60.265, 12.457, -150.061, 74.915, -188.524]
  Call Extruder(8897.852)
  MoveL 858 to (24.12, -11.61, 45) mm, rotated rx -180 ry 0 rz -180 deg; joints [29.229, 60.835, 11.041, -149.513, 74.249, -189.08]
  Call Extruder(8907.217)
  MoveL 859 to (26.09, -5.96, 45) mm, rotated rx 180 ry 0 rz 180 deg; joints [29.796, 61.336, 9.81, -148.822, 73.714, -189.63]
  Call Extruder(8916.582)
  MoveL 860 to (26.77, 0, 45) mm, rotated rx -180 ry 0 rz -180 deg; joints [30.482, 61.741, 8.824, -148.029, 73.336, -190.148]
  Call Extruder(8925.947)
  MoveL 861 to (26.09, 5.96, 45) mm, rotated rx 180 ry 0 rz -180 deg; joints [31.252, 62.026, 8.134, -147.171, 73.133, -190.603]
  Call Extruder(8935.312)
  MoveL 862 to (24.11, 11.61, 45) mm, rotated rx -180 ry 0 rz -180 deg; joints [32.076, 62.175, 7.774, -146.291, 73.111, -190.969]
  Call Extruder(8944.677)
  MoveL 863 to (20.93, 16.69, 45) mm, rotated rx 180 ry 0 rz -180 deg; joints [32.917, 62.179, 7.763, -145.427, 73.268, -191.222]
  Call Extruder(8954.042)
  MoveL 864 to (16.69, 20.93, 45) mm, rotated rx 180 ry 0 rz -180 deg; joints [33.742, 62.039, 8.103, -144.617, 73.592, -191.344]
  Call Extruder(8963.407)
  MoveL 865 to (11.61, 24.12, 45) mm, rotated rx 180 ry 0 rz 180 deg; joints [34.517, 61.761, 8.775, -143.893, 74.065, -191.324]
  Call Extruder(8972.772)
  MoveL 866 to (5.96, 26.09, 45) mm, rotated rx -180 ry 0 rz -180 deg; joints [35.208, 61.363, 9.745, -143.284, 74.66, -191.162]
  Call Extruder(8982.137)
  MoveL 867 to (0, 26.77, 45) mm, rotated rx 180 ry 0 rz -180 deg; joints [35.784, 60.867, 10.963, -142.815, 75.347, -190.863]
  Call Extruder(8991.502)
  MoveL 868 to (-5.96, 26.09, 45) mm, rotated rx 180 ry 0 rz -180 deg; joints [36.214, 60.3, 12.37, -142.509, 76.094, -190.446]
  Call Extruder(9000.867)
  MoveL 869 to (-11.61, 24.12, 45) mm, rotated rx 180 ry 0 rz -180 deg; joints [36.473, 59.694, 13.893, -142.38, 76.867, -189.932]
  Call Extruder(9010.232)
  MoveL 870 to (-16.69, 20.93, 45) mm, rotated rx 180 ry 0 rz 180 deg; joints [36.542, 59.079, 15.459, -142.443, 77.632, -189.353]
  Call Extruder(9019.597)
  MoveL 871 to (-20.93, 16.69, 45) mm, rotated rx 180 ry 0 rz 180 deg; joints [36.407, 58.487, 16.989, -142.7, 78.356, -188.741]
  Call Extruder(9028.962)
  MoveL 872 to (-24.12, 11.61, 45) mm, rotated rx 180 ry 0 rz -180 deg; joints [36.065, 57.946, 18.409, -143.151, 79.006, -188.134]
  Call Extruder(9038.326)
  MoveL 873 to (-26.09, 5.96, 45) mm, rotated rx -180 ry 0 rz -180 deg; joints [35.528, 57.481, 19.646, -143.78, 79.553, -187.565]
  Call Extruder(9047.692)
  MoveL 874 to (-26.77, 0, 45) mm, rotated rx 180 ry 0 rz 180 deg; joints [34.817, 57.113, 20.637, -144.562, 79.969, -187.067]
  Call Extruder(9052.480)
  MoveL 875 to (-26.42, -3.05, 45) mm, rotated rx 180 ry 0 rz -180 deg; joints [34.385, 56.981, 20.996, -145.02, 80.101, -186.859]
  Set speed (130.0 mm/s)
  MoveL 876 to (-41.86, -6.29, 45) mm, rotated rx -180 ry 0 rz -180 deg; joints [35.393, 55.712, 24.532, -144.212, 82.06, -185.687]
  Call Extruder(9057.478)
  Set speed (60.0 mm/s)
  MoveL 877 to (-41.51, -9.47, 45) mm, rotated rx -180 ry 0 rz 180 deg; joints [34.924, 55.584, 24.9, -144.702, 82.209, -185.482]
  Call Extruder(9072.374)
  MoveL 878 to (-38.36, -18.47, 45) mm, rotated rx 180 ry 0 rz 180 deg; joints [33.373, 55.382, 25.483, -146.29, 82.381, -185.055]
  Call Extruder(9087.270)
  MoveL 879 to (-33.29, -26.54, 45) mm, rotated rx 180 ry 0 rz 180 deg; joints [31.763, 55.376, 25.5, -147.909, 82.251, -184.833]
  Call Extruder(9102.165)
  MoveL 880 to (-26.54, -33.29, 45) mm, rotated rx 180 ry 0 rz 180 deg; joints [30.206, 55.566, 24.949, -149.45, 81.813, -184.804]
  Call Extruder(9117.061)
  MoveL 881 to (-18.47, -38.36, 45) mm, rotated rx 180 ry 0 rz -180 deg; joints [28.808, 55.948, 23.863, -150.806, 81.082, -184.95]
  Call Extruder(9131.957)
  MoveL 882 to (-9.47, -41.51, 45) mm, rotated rx -180 ry 0 rz 180 deg; joints [27.654, 56.506, 22.299, -151.891, 80.098, -185.248]
  Call Extruder(9146.853)
  MoveL 883 to (0, -42.57, 45) mm, rotated rx 180 ry 0 rz 180 deg; joints [26.805, 57.222, 20.343, -152.644, 78.919, -185.679]
  Call Extruder(9149.380)
  MoveL 884 to (1.61, -42.39, 45) mm, rotated rx 180 ry 0 rz -180 deg; joints [26.716, 57.362, 19.965, -152.713, 78.699, -185.772]
  Call Extruder(9161.749)
  MoveL 885 to (9.47, -41.5, 45) mm, rotated rx 180 ry 0 rz -180 deg; joints [26.29, 58.065, 18.094, -153.034, 77.615, -186.228]
  Call Extruder(9176.644)
  MoveL 886 to (18.47, -38.36, 45) mm, rotated rx 180 ry 0 rz 180 deg; joints [26.114, 58.999, 15.665, -153.056, 76.262, -186.883]
  Call Extruder(9191.540)
  MoveL 887 to (26.54, -33.28, 45) mm, rotated rx 180 ry 0 rz -180 deg; joints [26.262, 59.979, 13.174, -152.728, 74.936, -187.631]
  Call Extruder(9206.436)
  MoveL 888 to (33.28, -26.54, 45) mm, rotated rx 180 ry 0 rz -180 deg; joints [26.703, 60.956, 10.743, -152.085, 73.709, -188.453]
  Call Extruder(9221.332)
  MoveL 889 to (38.36, -18.47, 45) mm, rotated rx -180 ry 0 rz -180 deg; joints [27.4, 61.879, 8.489, -151.174, 72.645, -189.323]
  Call Extruder(9236.228)
  MoveL 890 to (41.5, -9.47, 45) mm, rotated rx 180 ry 0 rz 180 deg; joints [28.309, 62.696, 6.523, -150.053, 71.798, -190.202]
  Call Extruder(9251.123)
  MoveL 891 to (42.57, 0, 45) mm, rotated rx 180 ry 0 rz 180 deg; joints [29.382, 63.36, 4.945, -148.784, 71.209, -191.045]
  Call Extruder(9266.019)
  MoveL 892 to (41.5, 9.47, 45) mm, rotated rx -180 ry 0 rz -180 deg; joints [30.575, 63.829, 3.838, -147.433, 70.904, -191.803]
  Call Extruder(9280.915)
  MoveL 893 to (38.36, 18.47, 45) mm, rotated rx -180 ry 0 rz -180 deg; joints [31.839, 64.076, 3.259, -146.062, 70.892, -192.423]
  Call Extruder(9295.811)
  MoveL 894 to (33.28, 26.54, 45) mm, rotated rx 180 ry 0 rz -180 deg; joints [33.128, 64.083, 3.243, -144.73, 71.166, -192.861]
  Call Extruder(9310.707)
  MoveL 895 to (26.54, 33.29, 45) mm, rotated rx -180 ry 0 rz 180 deg; joints [34.394, 63.85, 3.788, -143.49, 71.704, -193.082]
  Call Extruder(9325.603)
  MoveL 896 to (18.47, 38.36, 45) mm, rotated rx -180 ry 0 rz 180 deg; joints [35.592, 63.393, 4.866, -142.384, 72.47, -193.067]
  Call Extruder(9340.498)
  MoveL 897 to (9.47, 41.5, 45) mm, rotated rx -180 ry 0 rz 180 deg; joints [36.675, 62.74, 6.419, -141.451, 73.42, -192.81]
  Call Extruder(9355.394)
  MoveL 898 to (0, 42.57, 45) mm, rotated rx 180 ry 0 rz -180 deg; joints [37.594, 61.931, 8.364, -140.723, 74.504, -192.325]
  Call Extruder(9370.290)
  MoveL 899 to (-9.47, 41.5, 45) mm, rotated rx 180 ry 0 rz 180 deg; joints [38.304, 61.013, 10.605, -140.228, 75.672, -191.639]
  Call Extruder(9385.186)
  MoveL 900 to (-18.47, 38.36, 45) mm, rotated rx 180 ry 0 rz -180 deg; joints [38.762, 60.037, 13.029, -139.992, 76.872, -190.793]
  Call Extruder(9400.081)
  MoveL 901 to (-26.54, 33.28, 45) mm, rotated rx 180 ry 0 rz 180 deg; joints [38.928, 59.056, 15.519, -140.04, 78.058, -189.836]
  Call Extruder(9414.977)
  MoveL 902 to (-33.29, 26.54, 45) mm, rotated rx -180 ry 0 rz 180 deg; joints [38.772, 58.118, 17.955, -140.391, 79.184, -188.827]
  Call Extruder(9429.873)
  MoveL 903 to (-38.36, 18.47, 45) mm, rotated rx 180 ry 0 rz 180 deg; joints [38.277, 57.268, 20.218, -141.051, 80.206, -187.829]
  Call Extruder(9444.769)
  MoveL 904 to (-41.51, 9.47, 45) mm, rotated rx -180 ry 0 rz 180 deg; joints [37.447, 56.544, 22.194, -142.014, 81.081, -186.903]
  Call Extruder(9459.665)
  MoveL 905 to (-42.57, 0, 45) mm, rotated rx 180 ry 0 rz 180 deg; joints [36.31, 55.976, 23.783, -143.25, 81.763, -186.106]
  Call Extruder(9467.219)
  MoveL 906 to (-42.03, -4.8, 45) mm, rotated rx 180 ry 0 rz -180 deg; joints [35.612, 55.774, 24.357, -143.983, 81.99, -185.785]
  Set speed (130.0 mm/s)
  MoveL 907 to (-54.1, -7.67, 45) mm, rotated rx 180 ry 0 rz -180 deg; joints [36.421, 54.839, 27.075, -143.305, 83.501, -184.821]
  Call Extruder(9471.292)
  Set speed (30.0 mm/s)
  MoveL 908 to (-53.59, -12.23, 45) mm, rotated rx 180 ry 0 rz 180 deg; joints [35.732, 54.662, 27.606, -144.02, 83.73, -184.534]
  Call Extruder(9482.222)
  MoveL 909 to (-49.52, -23.85, 45) mm, rotated rx -180 ry 0 rz -180 deg; joints [33.663, 54.41, 28.368, -146.126, 83.993, -184.018]
  Call Extruder(9493.152)
  MoveL 910 to (-42.98, -34.27, 45) mm, rotated rx 180 ry 0 rz -180 deg; joints [31.506, 54.402, 28.39, -148.292, 83.859, -183.781]
  Call Extruder(9504.082)
  MoveL 911 to (-34.27, -42.98, 45) mm, rotated rx 180 ry 0 rz -180 deg; joints [29.427, 54.64, 27.671, -150.351, 83.308, -183.795]
  Call Extruder(9515.012)
  MoveL 912 to (-23.85, -49.53, 45) mm, rotated rx -180 ry 0 rz -180 deg; joints [27.581, 55.117, 26.254, -152.151, 82.358, -184.019]
  Call Extruder(9525.942)
  MoveL 913 to (-12.23, -53.59, 45) mm, rotated rx 180 ry 0 rz 180 deg; joints [26.087, 55.822, 24.22, -153.568, 81.065, -184.415]
  Call Extruder(9536.873)
  MoveL 914 to (0, -54.97, 45) mm, rotated rx 180 ry 0 rz 180 deg; joints [25.019, 56.73, 21.682, -154.526, 79.513, -184.956]
  Call Extruder(9539.542)
  MoveL 915 to (2.99, -54.63, 45) mm, rotated rx 180 ry 0 rz 180 deg; joints [24.865, 56.987, 20.98, -154.646, 79.097, -185.122]
  Call Extruder(9547.803)
  MoveL 916 to (12.23, -53.59, 45) mm, rotated rx 180 ry 0 rz 180 deg; joints [24.406, 57.808, 18.772, -154.992, 77.799, -185.63]
  Call Extruder(9558.733)
  MoveL 917 to (23.85, -49.53, 45) mm, rotated rx -180 ry 0 rz -180 deg; joints [24.239, 59.011, 15.635, -154.972, 76.028, -186.432]
  Call Extruder(9569.663)
  MoveL 918 to (34.27, -42.98, 45) mm, rotated rx -180 ry 0 rz -180 deg; joints [24.487, 60.28, 12.42, -154.497, 74.298, -187.356]
  Call Extruder(9580.593)
  MoveL 919 to (42.98, -34.27, 45) mm, rotated rx 180 ry 0 rz 180 deg; joints [25.101, 61.554, 9.278, -153.621, 72.703, -188.388]
  Call Extruder(9591.524)
  MoveL 920 to (49.52, -23.85, 45) mm, rotated rx 180 ry 0 rz -180 deg; joints [26.025, 62.764, 6.361, -152.41, 71.325, -189.499]
  Call Extruder(9602.454)
  MoveL 921 to (53.59, -12.23, 45) mm, rotated rx -180 ry 0 rz -180 deg; joints [27.2, 63.841, 3.81, -150.94, 70.233, -190.643]
  Call Extruder(9613.384)
  MoveL 922 to (54.97, 0, 45) mm, rotated rx -180 ry 0 rz -180 deg; joints [28.57, 64.721, 1.756, -149.294, 69.481, -191.759]
  Call Extruder(9624.314)
  MoveL 923 to (53.59, 12.23, 45) mm, rotated rx 180 ry 0 rz -180 deg; joints [30.077, 65.346, 0.31, -147.558, 69.102, -192.775]
  Call Extruder(9635.244)
  MoveL 924 to (49.53, 23.85, 45) mm, rotated rx 180 ry 0 rz -180 deg; joints [31.665, 65.675, -0.445, -145.813, 69.108, -193.617]
  Call Extruder(9646.175)
  MoveL 925 to (42.98, 34.27, 45) mm, rotated rx 180 ry 0 rz -180 deg; joints [33.282, 65.684, -0.467, -144.132, 69.487, -194.218]
  Call Extruder(9657.105)
  MoveL 926 to (34.27, 42.98, 45) mm, rotated rx 180 ry 0 rz 180 deg; joints [34.874, 65.374, 0.246, -142.578, 70.205, -194.527]
  Call Extruder(9668.035)
  MoveL 927 to (23.85, 49.52, 45) mm, rotated rx -180 ry 0 rz 180 deg; joints [36.387, 64.765, 1.653, -141.199, 71.212, -194.518]
  Call Extruder(9678.965)
  MoveL 928 to (12.23, 53.59, 45) mm, rotated rx 180 ry 0 rz 180 deg; joints [37.766, 63.899, 3.674, -140.033, 72.447, -194.185]
  Call Extruder(9689.896)
  MoveL 929 to (0, 54.97, 45) mm, rotated rx -180 ry 0 rz -180 deg; joints [38.954, 62.832, 6.199, -139.114, 73.842, -193.547]
  Call Extruder(9700.826)
  MoveL 930 to (-12.23, 53.59, 45) mm, rotated rx 180 ry 0 rz -180 deg; joints [39.895, 61.628, 9.099, -138.472, 75.331, -192.641]
  Call Extruder(9711.756)
  MoveL 931 to (-23.85, 49.52, 45) mm, rotated rx -180 ry 0 rz -180 deg; joints [40.528, 60.356, 12.231, -138.14, 76.852, -191.519]
  Call Extruder(9722.686)
  MoveL 932 to (-34.27, 42.98, 45) mm, rotated rx -180 ry 0 rz -180 deg; joints [40.799, 59.084, 15.446, -138.152, 78.351, -190.25]
  Call Extruder(9733.616)
  MoveL 933 to (-42.98, 34.27, 45) mm, rotated rx -180 ry 0 rz 180 deg; joints [40.659, 57.876, 18.593, -138.543, 79.776, -188.911]
  Call Extruder(9744.547)
  MoveL 934 to (-49.53, 23.85, 45) mm, rotated rx -180 ry 0 rz -180 deg; joints [40.072, 56.789, 21.52, -139.335, 81.08, -187.588]
  Call Extruder(9755.477)
  MoveL 935 to (-53.59, 12.23, 45) mm, rotated rx 180 ry 0 rz 180 deg; joints [39.031, 55.87, 24.083, -140.536, 82.211, -186.366]
  Call Extruder(9766.407)
  MoveL 936 to (-54.97, 0, 45) mm, rotated rx 180 ry 0 rz 180 deg; joints [37.56, 55.153, 26.15, -142.119, 83.115, -185.328]
  Call Extruder(9771.933)
  MoveL 937 to (-54.27, -6.18, 45) mm, rotated rx 180 ry 0 rz -180 deg; joints [36.644, 54.899, 26.898, -143.073, 83.426, -184.917]
  Set speed (130.0 mm/s)
  MoveL 938 to (-49.9, -9.51, 45) mm, rotated rx 180 ry 0 rz -180 deg; joints [35.741, 55.023, 26.53, -143.962, 83.153, -184.958]
  MoveL 939 to (2.97, -12.99, 45) mm, rotated rx 180 ry 0 rz 180 deg; joints [30.614, 58.838, 16.079, -148.498, 77.059, -187.815]
  Call Extruder(9776.596)
  Set speed (80.0 mm/s)
  MoveL 940 to (5.78, -12.01, 45) mm, rotated rx 180 ry 0 rz -180 deg; joints [30.526, 59.134, 15.319, -148.531, 76.651, -188.043]
  Call Extruder(9781.260)
  MoveL 941 to (8.31, -10.42, 45) mm, rotated rx -180 ry 0 rz -180 deg; joints [30.538, 59.439, 14.539, -148.459, 76.248, -188.301]
  Call Extruder(9785.924)
  MoveL 942 to (10.42, -8.31, 45) mm, rotated rx -180 ry 0 rz -180 deg; joints [30.649, 59.739, 13.778, -148.286, 75.872, -188.578]
  Call Extruder(9790.588)
  MoveL 943 to (12.01, -5.78, 45) mm, rotated rx -180 ry 0 rz -180 deg; joints [30.85, 60.019, 13.073, -148.024, 75.542, -188.86]
  Call Extruder(9795.251)
  MoveL 944 to (12.99, -2.97, 45) mm, rotated rx 180 ry 0 rz -180 deg; joints [31.131, 60.264, 12.461, -147.687, 75.274, -189.134]
  Call Extruder(9799.915)
  MoveL 945 to (13.33, 0, 45) mm, rotated rx 180 ry 0 rz -180 deg; joints [31.476, 60.46, 11.971, -147.292, 75.082, -189.387]
  Call Extruder(9804.579)
  MoveL 946 to (12.99, 2.97, 45) mm, rotated rx -180 ry 0 rz -180 deg; joints [31.869, 60.598, 11.628, -146.861, 74.975, -189.606]
  Call Extruder(9809.243)
  MoveL 947 to (12.01, 5.78, 45) mm, rotated rx -180 ry 0 rz 180 deg; joints [32.292, 60.67, 11.449, -146.414, 74.957, -189.779]
  Call Extruder(9813.906)
  MoveL 948 to (10.42, 8.31, 45) mm, rotated rx 180 ry 0 rz 180 deg; joints [32.725, 60.672, 11.444, -145.972, 75.029, -189.895]
  Call Extruder(9818.570)
  MoveL 949 to (8.31, 10.42, 45) mm, rotated rx 180 ry 0 rz -180 deg; joints [33.149, 60.605, 11.613, -145.555, 75.185, -189.948]
  Call Extruder(9823.234)
  MoveL 950 to (5.78, 12.01, 45) mm, rotated rx 180 ry 0 rz -180 deg; joints [33.544, 60.47, 11.946, -145.182, 75.417, -189.933]
  Call Extruder(9827.898)
  MoveL 951 to (2.97, 13, 45) mm, rotated rx 180 ry 0 rz 180 deg; joints [33.893, 60.277, 12.428, -144.87, 75.713, -189.85]
  Call Extruder(9832.562)
  MoveL 952 to (0, 13.33, 45) mm, rotated rx -180 ry 0 rz 180 deg; joints [34.177, 60.035, 13.035, -144.633, 76.059, -189.704]
  Call Extruder(9837.226)
  MoveL 953 to (-2.97, 13, 45) mm, rotated rx 180 ry 0 rz 180 deg; joints [34.384, 59.757, 13.735, -144.484, 76.437, -189.502]
  Call Extruder(9841.889)
  MoveL 954 to (-5.78, 12.01, 45) mm, rotated rx -180 ry 0 rz -180 deg; joints [34.5, 59.457, 14.493, -144.429, 76.83, -189.255]
  Call Extruder(9846.553)
  MoveL 955 to (-8.31, 10.42, 45) mm, rotated rx 180 ry 0 rz 180 deg; joints [34.518, 59.151, 15.273, -144.474, 77.219, -188.976]
  Call Extruder(9851.217)
  MoveL 956 to (-10.42, 8.31, 45) mm, rotated rx -180 ry 0 rz -180 deg; joints [34.436, 58.855, 16.035, -144.618, 77.585, -188.681]
  Call Extruder(9855.881)
  MoveL 957 to (-12.01, 5.78, 45) mm, rotated rx 180 ry 0 rz 180 deg; joints [34.254, 58.582, 16.741, -144.856, 77.912, -188.386]
  Call Extruder(9860.544)
  MoveL 958 to (-13, 2.97, 45) mm, rotated rx -180 ry 0 rz -180 deg; joints [33.981, 58.347, 17.355, -145.178, 78.183, -188.107]
  Call Extruder(9865.208)
  MoveL 959 to (-13.33, 0, 45) mm, rotated rx 180 ry 0 rz -180 deg; joints [33.63, 58.159, 17.846, -145.57, 78.384, -187.859]
  Call Extruder(9869.872)
  MoveL 960 to (-13, -2.97, 45) mm, rotated rx 180 ry 0 rz 180 deg; joints [33.218, 58.028, 18.191, -146.011, 78.505, -187.653]
  Call Extruder(9874.536)
  MoveL 961 to (-12.01, -5.78, 45) mm, rotated rx -180 ry 0 rz -180 deg; joints [32.767, 57.96, 18.37, -146.479, 78.538, -187.499]
  Call Extruder(9879.199)
  MoveL 962 to (-10.42, -8.31, 45) mm, rotated rx 180 ry 0 rz -180 deg; joints [32.302, 57.958, 18.375, -146.95, 78.48, -187.404]
  Call Extruder(9883.863)
  MoveL 963 to (-8.31, -10.42, 45) mm, rotated rx 180 ry 0 rz 180 deg; joints [31.85, 58.023, 18.206, -147.396, 78.334, -187.37]
  Call Extruder(9888.527)
  MoveL 964 to (-5.78, -12.01, 45) mm, rotated rx 180 ry 0 rz 180 deg; joints [31.435, 58.15, 17.871, -147.793, 78.105, -187.397]
  Call Extruder(9893.191)
  MoveL 965 to (-2.97, -13, 45) mm, rotated rx -180 ry 0 rz 180 deg; joints [31.079, 58.334, 17.387, -148.12, 77.806, -187.484]
  Call Extruder(9897.855)
  MoveL 966 to (0, -13.33, 45) mm, rotated rx 180 ry 0 rz 180 deg; joints [30.801, 58.567, 16.78, -148.359, 77.451, -187.626]
  Call Extruder(9902.518)
  MoveL 967 to (2.97, -12.99, 45) mm, rotated rx 180 ry 0 rz 180 deg; joints [30.614, 58.838, 16.079, -148.498, 77.059, -187.815]
  Set speed (130.0 mm/s)
  MoveL 968 to (2.97, -12.99, 50) mm, rotated rx -180 ry 0 rz -180 deg; joints [30.614, 57.903, 16.528, -148.439, 76.645, -188.076]
  MoveL 969 to (-26.25, -4.54, 50) mm, rotated rx 180 ry 0 rz -180 deg; joints [34.172, 55.948, 21.622, -145.193, 79.742, -187.058]
  Call Extruder(9904.751)
  Set speed (60.0 mm/s)
  MoveL 970 to (-26.09, -5.96, 50) mm, rotated rx -180 ry 0 rz -180 deg; joints [33.969, 55.886, 21.786, -145.409, 79.801, -186.962]
  Call Extruder(9914.116)
  MoveL 971 to (-24.12, -11.61, 50) mm, rotated rx 180 ry 0 rz 180 deg; joints [33.033, 55.751, 22.149, -146.376, 79.879, -186.665]
  Call Extruder(9923.481)
  MoveL 972 to (-20.93, -16.69, 50) mm, rotated rx 180 ry 0 rz 180 deg; joints [32.066, 55.748, 22.159, -147.353, 79.774, -186.489]
  Call Extruder(9932.846)
  MoveL 973 to (-16.69, -20.93, 50) mm, rotated rx 180 ry 0 rz -180 deg; joints [31.126, 55.875, 21.817, -148.281, 79.486, -186.435]
  Call Extruder(9942.211)
  MoveL 974 to (-11.61, -24.12, 50) mm, rotated rx -180 ry 0 rz -180 deg; joints [30.272, 56.128, 21.14, -149.103, 79.028, -186.498]
  Call Extruder(9951.576)
  MoveL 975 to (-5.96, -26.09, 50) mm, rotated rx 180 ry 0 rz 180 deg; joints [29.552, 56.497, 20.164, -149.771, 78.422, -186.67]
  Call Extruder(9960.941)
  MoveL 976 to (0, -26.77, 50) mm, rotated rx 180 ry 0 rz 180 deg; joints [29.003, 56.965, 18.938, -150.248, 77.701, -186.942]
  Call Extruder(9970.306)
  MoveL 977 to (5.96, -26.09, 50) mm, rotated rx 180 ry 0 rz 180 deg; joints [28.65, 57.512, 17.527, -150.511, 76.905, -187.301]
  Call Extruder(9979.671)
  MoveL 978 to (11.61, -24.11, 50) mm, rotated rx 180 ry 0 rz -180 deg; joints [28.503, 58.111, 16, -150.552, 76.079, -187.735]
  Call Extruder(9989.036)
  MoveL 979 to (16.69, -20.93, 50) mm, rotated rx -180 ry 0 rz 180 deg; joints [28.559, 58.735, 14.434, -150.375, 75.267, -188.229]
  Call Extruder(9998.401)
  MoveL 980 to (20.93, -16.69, 50) mm, rotated rx -180 ry 0 rz -180 deg; joints [28.808, 59.352, 12.906, -149.998, 74.513, -188.765]
  Call Extruder(10007.766)
  MoveL 981 to (24.12, -11.61, 50) mm, rotated rx 180 ry 0 rz 180 deg; joints [29.229, 59.929, 11.491, -149.446, 73.855, -189.322]
  Call Extruder(10017.131)
  MoveL 982 to (26.09, -5.96, 50) mm, rotated rx 180 ry 0 rz 180 deg; joints [29.796, 60.437, 10.26, -148.753, 73.329, -189.874]
  Call Extruder(10026.496)
  MoveL 983 to (26.77, 0, 50) mm, rotated rx 180 ry 0 rz -180 deg; joints [30.482, 60.846, 9.274, -147.957, 72.959, -190.394]
  Call Extruder(10035.861)
  MoveL 984 to (26.09, 5.96, 50) mm, rotated rx -180 ry 0 rz 180 deg; joints [31.252, 61.134, 8.584, -147.098, 72.762, -190.853]
  Call Extruder(10045.226)
  MoveL 985 to (24.11, 11.61, 50) mm, rotated rx 180 ry 0 rz -180 deg; joints [32.076, 61.285, 8.224, -146.216, 72.745, -191.224]
  Call Extruder(10054.591)
  MoveL 986 to (20.93, 16.69, 50) mm, rotated rx -180 ry 0 rz -180 deg; joints [32.917, 61.289, 8.214, -145.351, 72.906, -191.483]
  Call Extruder(10063.956)
  MoveL 987 to (16.69, 20.93, 50) mm, rotated rx 180 ry 0 rz -180 deg; joints [33.742, 61.147, 8.553, -144.541, 73.233, -191.611]
  Call Extruder(10073.321)
  MoveL 988 to (11.61, 24.12, 50) mm, rotated rx 180 ry 0 rz 180 deg; joints [34.517, 60.866, 9.225, -143.817, 73.706, -191.597]
  Call Extruder(10082.685)
  MoveL 989 to (5.96, 26.09, 50) mm, rotated rx -180 ry 0 rz -180 deg; joints [35.208, 60.464, 10.194, -143.209, 74.299, -191.441]
  Call Extruder(10092.051)
  MoveL 990 to (0, 26.77, 50) mm, rotated rx -180 ry 0 rz 180 deg; joints [35.784, 59.961, 11.412, -142.742, 74.983, -191.149]
  Call Extruder(10101.416)
  MoveL 991 to (-5.96, 26.09, 50) mm, rotated rx 180 ry 0 rz -180 deg; joints [36.214, 59.387, 12.818, -142.438, 75.726, -190.737]
  Call Extruder(10110.780)
  MoveL 992 to (-11.61, 24.12, 50) mm, rotated rx 180 ry 0 rz 180 deg; joints [36.473, 58.772, 14.342, -142.312, 76.492, -190.229]
  Call Extruder(10120.145)
  MoveL 993 to (-16.69, 20.93, 50) mm, rotated rx 180 ry 0 rz 180 deg; joints [36.542, 58.148, 15.908, -142.377, 77.25, -189.654]
  Call Extruder(10129.511)
  MoveL 994 to (-20.93, 16.69, 50) mm, rotated rx -180 ry 0 rz -180 deg; joints [36.407, 57.546, 17.44, -142.638, 77.965, -189.045]
  Call Extruder(10138.875)
  MoveL 995 to (-24.12, 11.61, 50) mm, rotated rx 180 ry 0 rz -180 deg; joints [36.065, 56.995, 18.86, -143.091, 78.607, -188.439]
  Call Extruder(10148.240)
  MoveL 996 to (-26.09, 5.96, 50) mm, rotated rx 180 ry 0 rz -180 deg; joints [35.528, 56.522, 20.098, -143.723, 79.144, -187.87]
  Call Extruder(10157.605)
  MoveL 997 to (-26.77, 0, 50) mm, rotated rx 180 ry 0 rz 180 deg; joints [34.817, 56.147, 21.09, -144.508, 79.551, -187.369]
  Call Extruder(10162.394)
  MoveL 998 to (-26.42, -3.05, 50) mm, rotated rx 180 ry 0 rz -180 deg; joints [34.385, 56.012, 21.449, -144.968, 79.679, -187.159]
  Set speed (130.0 mm/s)
  MoveL 999 to (-41.86, -6.29, 50) mm, rotated rx 180 ry 0 rz 180 deg; joints [35.393, 54.715, 24.99, -144.167, 81.623, -186.005]
  Call Extruder(10167.392)
  Set speed (60.0 mm/s)
  MoveL 1000 to (-41.51, -9.47, 50) mm, rotated rx 180 ry 0 rz 180 deg; joints [34.924, 54.584, 25.359, -144.658, 81.768, -185.798]
  Call Extruder(10182.288)
  MoveL 1001 to (-38.36, -18.47, 50) mm, rotated rx -180 ry 0 rz 180 deg; joints [33.373, 54.377, 25.943, -146.248, 81.928, -185.361]
  Call Extruder(10197.183)
  MoveL 1002 to (-33.29, -26.54, 50) mm, rotated rx 180 ry 0 rz 180 deg; joints [31.763, 54.371, 25.96, -147.869, 81.79, -185.125]
  Call Extruder(10212.079)
  MoveL 1003 to (-26.54, -33.28, 50) mm, rotated rx 180 ry 0 rz 180 deg; joints [30.206, 54.566, 25.409, -149.409, 81.347, -185.083]
  Call Extruder(10226.975)
  MoveL 1004 to (-18.47, -38.36, 50) mm, rotated rx 180 ry 0 rz -180 deg; joints [28.808, 54.956, 24.32, -150.764, 80.616, -185.214]
  Call Extruder(10241.871)
  MoveL 1005 to (-9.47, -41.5, 50) mm, rotated rx 180 ry 0 rz 180 deg; joints [27.654, 55.528, 22.754, -151.847, 79.636, -185.499]
  Call Extruder(10256.767)
  MoveL 1006 to (0, -42.57, 50) mm, rotated rx -180 ry 0 rz 180 deg; joints [26.805, 56.258, 20.796, -152.597, 78.465, -185.919]
  Call Extruder(10259.950)
  MoveL 1007 to (2.02, -42.34, 50) mm, rotated rx 180 ry 0 rz 180 deg; joints [26.692, 56.438, 20.319, -152.683, 78.19, -186.035]
  Call Extruder(10271.663)
  MoveL 1008 to (9.47, -41.5, 50) mm, rotated rx 180 ry 0 rz -180 deg; joints [26.29, 57.117, 18.545, -152.983, 77.172, -186.459]
  Call Extruder(10286.558)
  MoveL 1009 to (18.47, -38.36, 50) mm, rotated rx 180 ry 0 rz 180 deg; joints [26.114, 58.066, 16.114, -153.001, 75.831, -187.109]
  Call Extruder(10301.454)
  MoveL 1010 to (26.54, -33.28, 50) mm, rotated rx 180 ry 0 rz 180 deg; joints [26.262, 59.061, 13.623, -152.669, 74.52, -187.854]
  Call Extruder(10316.350)
  MoveL 1011 to (33.28, -26.54, 50) mm, rotated rx -180 ry 0 rz 180 deg; joints [26.703, 60.052, 11.192, -152.021, 73.307, -188.676]
  Call Extruder(10331.246)
  MoveL 1012 to (38.36, -18.47, 50) mm, rotated rx 180 ry 0 rz -180 deg; joints [27.4, 60.986, 8.939, -151.106, 72.257, -189.547]
  Call Extruder(10346.141)
  MoveL 1013 to (41.51, -9.47, 50) mm, rotated rx -180 ry 0 rz -180 deg; joints [28.309, 61.812, 6.975, -149.981, 71.423, -190.43]
  Call Extruder(10361.037)
  MoveL 1014 to (42.57, 0, 50) mm, rotated rx -180 ry 0 rz -180 deg; joints [29.382, 62.482, 5.398, -148.709, 70.846, -191.278]
  Call Extruder(10375.933)
  MoveL 1015 to (41.5, 9.47, 50) mm, rotated rx 180 ry 0 rz -180 deg; joints [30.575, 62.956, 4.292, -147.354, 70.551, -192.042]
  Call Extruder(10390.829)
  MoveL 1016 to (38.36, 18.47, 50) mm, rotated rx 180 ry 0 rz 180 deg; joints [31.839, 63.205, 3.715, -145.981, 70.547, -192.67]
  Call Extruder(10405.725)
  MoveL 1017 to (33.28, 26.54, 50) mm, rotated rx 180 ry 0 rz 180 deg; joints [33.128, 63.212, 3.698, -144.648, 70.826, -193.116]
  Call Extruder(10420.620)
  MoveL 1018 to (26.54, 33.29, 50) mm, rotated rx 180 ry 0 rz 180 deg; joints [34.394, 62.977, 4.243, -143.407, 71.367, -193.345]
  Call Extruder(10435.516)
  MoveL 1019 to (18.47, 38.36, 50) mm, rotated rx 180 ry 0 rz 180 deg; joints [35.592, 62.516, 5.319, -142.302, 72.134, -193.339]
  Call Extruder(10450.412)
  MoveL 1020 to (9.47, 41.51, 50) mm, rotated rx 180 ry 0 rz 180 deg; joints [36.675, 61.856, 6.87, -141.37, 73.082, -193.091]
  Call Extruder(10465.308)
  MoveL 1021 to (0, 42.57, 50) mm, rotated rx 180 ry 0 rz -180 deg; joints [37.594, 61.038, 8.814, -140.644, 74.162, -192.616]
  Call Extruder(10480.204)
  MoveL 1022 to (-9.47, 41.51, 50) mm, rotated rx 180 ry 0 rz 180 deg; joints [38.304, 60.109, 11.054, -140.152, 75.323, -191.94]
  Call Extruder(10495.099)
  MoveL 1023 to (-18.47, 38.36, 50) mm, rotated rx -180 ry 0 rz -180 deg; joints [38.762, 59.12, 13.478, -139.921, 76.514, -191.102]
  Call Extruder(10509.995)
  MoveL 1024 to (-26.54, 33.29, 50) mm, rotated rx 180 ry 0 rz 180 deg; joints [38.928, 58.124, 15.968, -139.974, 77.689, -190.153]
  Call Extruder(10524.891)
  MoveL 1025 to (-33.29, 26.54, 50) mm, rotated rx 180 ry 0 rz 180 deg; joints [38.772, 57.171, 18.406, -140.329, 78.802, -189.15]
  Call Extruder(10539.787)
  MoveL 1026 to (-38.36, 18.47, 50) mm, rotated rx 180 ry 0 rz 180 deg; joints [38.277, 56.305, 20.67, -140.994, 79.81, -188.155]
  Call Extruder(10554.683)
  MoveL 1027 to (-41.51, 9.47, 50) mm, rotated rx 180 ry 0 rz -180 deg; joints [37.447, 55.566, 22.649, -141.962, 80.669, -187.229]
  Call Extruder(10569.578)
  MoveL 1028 to (-42.57, 0, 50) mm, rotated rx -180 ry 0 rz -180 deg; joints [36.31, 54.985, 24.241, -143.202, 81.336, -186.429]
  Call Extruder(10577.133)
  MoveL 1029 to (-42.03, -4.8, 50) mm, rotated rx 180 ry 0 rz -180 deg; joints [35.612, 54.778, 24.815, -143.937, 81.555, -186.104]
  Set speed (130.0 mm/s)
  MoveL 1030 to (-54.1, -7.67, 50) mm, rotated rx 180 ry 0 rz -180 deg; joints [36.421, 53.82, 27.538, -143.266, 83.056, -185.156]
  Call Extruder(10581.205)
  Set speed (30.0 mm/s)
  MoveL 1031 to (-53.59, -12.23, 50) mm, rotated rx -180 ry 0 rz 180 deg; joints [35.732, 53.638, 28.07, -143.982, 83.277, -184.865]
  Call Extruder(10592.135)
  MoveL 1032 to (-49.53, -23.85, 50) mm, rotated rx -180 ry 0 rz 180 deg; joints [33.663, 53.378, 28.834, -146.092, 83.524, -184.335]
  Call Extruder(10603.066)
  MoveL 1033 to (-42.98, -34.27, 50) mm, rotated rx 180 ry 0 rz 180 deg; joints [31.506, 53.371, 28.856, -148.258, 83.378, -184.08]
  Call Extruder(10613.996)
  MoveL 1034 to (-34.27, -42.98, 50) mm, rotated rx 180 ry 0 rz 180 deg; joints [29.427, 53.615, 28.135, -150.318, 82.821, -184.074]
  Call Extruder(10624.926)
  MoveL 1035 to (-23.85, -49.53, 50) mm, rotated rx 180 ry 0 rz 180 deg; joints [27.581, 54.106, 26.715, -152.115, 81.871, -184.279]
  Call Extruder(10635.856)
  MoveL 1036 to (-12.23, -53.59, 50) mm, rotated rx 180 ry 0 rz 180 deg; joints [26.087, 54.827, 24.678, -153.53, 80.585, -184.657]
  Call Extruder(10646.786)
  MoveL 1037 to (0, -54.97, 50) mm, rotated rx 180 ry 0 rz -180 deg; joints [25.019, 55.756, 22.137, -154.484, 79.043, -185.184]
  Call Extruder(10649.828)
  MoveL 1038 to (3.4, -54.58, 50) mm, rotated rx 180 ry 0 rz 180 deg; joints [24.844, 56.055, 21.334, -154.618, 78.573, -185.37]
  Call Extruder(10657.717)
  MoveL 1039 to (12.23, -53.59, 50) mm, rotated rx -180 ry 0 rz 180 deg; joints [24.406, 56.856, 19.224, -154.945, 77.345, -185.848]
  Call Extruder(10668.647)
  MoveL 1040 to (23.85, -49.52, 50) mm, rotated rx 180 ry 0 rz -180 deg; joints [24.239, 58.078, 16.084, -154.92, 75.59, -186.643]
  Call Extruder(10679.577)
  MoveL 1041 to (34.27, -42.98, 50) mm, rotated rx 180 ry 0 rz -180 deg; joints [24.487, 59.367, 12.869, -154.44, 73.879, -187.564]
  Call Extruder(10690.507)
  MoveL 1042 to (42.98, -34.27, 50) mm, rotated rx 180 ry 0 rz -180 deg; joints [25.101, 60.657, 9.728, -153.558, 72.302, -188.597]
  Call Extruder(10701.438)
  MoveL 1043 to (49.52, -23.85, 50) mm, rotated rx 180 ry 0 rz 180 deg; joints [26.025, 61.88, 6.812, -152.341, 70.942, -189.711]
  Call Extruder(10712.368)
  MoveL 1044 to (53.59, -12.23, 50) mm, rotated rx 180 ry 0 rz -180 deg; joints [27.2, 62.968, 4.264, -150.866, 69.867, -190.86]
  Call Extruder(10723.298)
  MoveL 1045 to (54.97, 0, 50) mm, rotated rx 180 ry 0 rz 180 deg; joints [28.57, 63.855, 2.213, -149.215, 69.13, -191.983]
  Call Extruder(10734.228)
  MoveL 1046 to (53.59, 12.23, 50) mm, rotated rx -180 ry 0 rz -180 deg; joints [30.077, 64.485, 0.77, -147.475, 68.763, -193.006]
  Call Extruder(10745.158)
  MoveL 1047 to (49.52, 23.85, 50) mm, rotated rx 180 ry 0 rz 180 deg; joints [31.665, 64.816, 0.016, -145.727, 68.779, -193.857]
  Call Extruder(10756.088)
  MoveL 1048 to (42.98, 34.27, 50) mm, rotated rx 180 ry 0 rz 180 deg; joints [33.282, 64.825, -0.006, -144.044, 69.165, -194.467]
  Call Extruder(10767.019)
  MoveL 1049 to (34.27, 42.98, 50) mm, rotated rx -180 ry 0 rz -180 deg; joints [34.874, 64.513, 0.706, -142.489, 69.887, -194.787]
  Call Extruder(10777.949)
  MoveL 1050 to (23.85, 49.53, 50) mm, rotated rx 180 ry 0 rz 180 deg; joints [36.387, 63.9, 2.111, -141.111, 70.895, -194.789]
  Call Extruder(10788.879)
  MoveL 1051 to (12.23, 53.59, 50) mm, rotated rx 180 ry 0 rz 180 deg; joints [37.766, 63.026, 4.128, -139.947, 72.127, -194.468]
  Call Extruder(10799.809)
  MoveL 1052 to (0, 54.97, 50) mm, rotated rx -180 ry 0 rz -180 deg; joints [38.954, 61.949, 6.651, -139.031, 73.516, -193.841]
  Call Extruder(10810.739)
  MoveL 1053 to (-12.23, 53.59, 50) mm, rotated rx -180 ry 0 rz -180 deg; joints [39.895, 60.731, 9.549, -138.393, 74.997, -192.947]
  Call Extruder(10821.670)
  MoveL 1054 to (-23.85, 49.52, 50) mm, rotated rx 180 ry 0 rz 180 deg; joints [40.528, 59.443, 12.68, -138.066, 76.507, -191.837]
  Call Extruder(10832.600)
  MoveL 1055 to (-34.27, 42.98, 50) mm, rotated rx 180 ry 0 rz 180 deg; joints [40.799, 58.153, 15.896, -138.085, 77.992, -190.579]
  Call Extruder(10843.530)
  MoveL 1056 to (-42.98, 34.27, 50) mm, rotated rx -180 ry 0 rz 180 deg; joints [40.659, 56.925, 19.044, -138.482, 79.401, -189.248]
  Call Extruder(10854.460)
  MoveL 1057 to (-49.53, 23.85, 50) mm, rotated rx 180 ry 0 rz -180 deg; joints [40.072, 55.816, 21.974, -139.281, 80.687, -187.93]
  Call Extruder(10865.390)
  MoveL 1058 to (-53.59, 12.23, 50) mm, rotated rx 180 ry 0 rz -180 deg; joints [39.031, 54.877, 24.541, -140.488, 81.798, -186.71]
  Call Extruder(10876.321)
  MoveL 1059 to (-54.97, 0, 50) mm, rotated rx 180 ry 0 rz -180 deg; joints [37.56, 54.142, 26.611, -142.077, 82.682, -185.668]
  Call Extruder(10881.846)
  MoveL 1060 to (-54.27, -6.18, 50) mm, rotated rx 180 ry 0 rz 180 deg; joints [36.644, 53.881, 27.361, -143.033, 82.983, -185.253]
  Set speed (130.0 mm/s)
  MoveL 1061 to (-49.9, -9.51, 50) mm, rotated rx -180 ry 0 rz -180 deg; joints [35.741, 54.009, 26.992, -143.921, 82.706, -185.285]
  MoveL 1062 to (2.97, -12.99, 50) mm, rotated rx -180 ry 0 rz -180 deg; joints [30.614, 57.903, 16.528, -148.439, 76.645, -188.076]
  Call Extruder(10886.510)
  Set speed (80.0 mm/s)
  MoveL 1063 to (5.78, -12.01, 50) mm, rotated rx -180 ry 0 rz -180 deg; joints [30.526, 58.203, 15.768, -148.471, 76.241, -188.302]
  Call Extruder(10891.173)
  MoveL 1064 to (8.31, -10.42, 50) mm, rotated rx 180 ry 0 rz 180 deg; joints [30.538, 58.513, 14.988, -148.397, 75.842, -188.559]
  Call Extruder(10895.838)
  MoveL 1065 to (10.42, -8.31, 50) mm, rotated rx 180 ry 0 rz -180 deg; joints [30.649, 58.818, 14.227, -148.223, 75.47, -188.834]
  Call Extruder(10900.501)
  MoveL 1066 to (12.01, -5.78, 50) mm, rotated rx 180 ry 0 rz 180 deg; joints [30.85, 59.102, 13.522, -147.959, 75.145, -189.116]
  Call Extruder(10905.165)
  MoveL 1067 to (12.99, -2.97, 50) mm, rotated rx 180 ry 0 rz -180 deg; joints [31.131, 59.35, 12.91, -147.62, 74.881, -189.391]
  Call Extruder(10909.829)
  MoveL 1068 to (13.33, 0, 50) mm, rotated rx 180 ry 0 rz -180 deg; joints [31.476, 59.549, 12.42, -147.225, 74.693, -189.646]
  Call Extruder(10914.493)
  MoveL 1069 to (12.99, 2.97, 50) mm, rotated rx 180 ry 0 rz -180 deg; joints [31.869, 59.689, 12.077, -146.793, 74.59, -189.867]
  Call Extruder(10919.156)
  MoveL 1070 to (12.01, 5.78, 50) mm, rotated rx 180 ry 0 rz -180 deg; joints [32.292, 59.762, 11.899, -146.345, 74.575, -190.042]
  Call Extruder(10923.820)
  MoveL 1071 to (10.42, 8.31, 50) mm, rotated rx -180 ry 0 rz 180 deg; joints [32.725, 59.764, 11.893, -145.902, 74.648, -190.161]
  Call Extruder(10928.484)
  MoveL 1072 to (8.31, 10.42, 50) mm, rotated rx 180 ry 0 rz 180 deg; joints [33.149, 59.695, 12.062, -145.485, 74.805, -190.217]
  Call Extruder(10933.148)
  MoveL 1073 to (5.78, 12.01, 50) mm, rotated rx -180 ry 0 rz -180 deg; joints [33.544, 59.559, 12.395, -145.112, 75.038, -190.206]
  Call Extruder(10937.811)
  MoveL 1074 to (2.97, 13, 50) mm, rotated rx 180 ry 0 rz -180 deg; joints [33.893, 59.363, 12.877, -144.801, 75.333, -190.126]
  Call Extruder(10942.475)
  MoveL 1075 to (0, 13.33, 50) mm, rotated rx 180 ry 0 rz 180 deg; joints [34.177, 59.118, 13.484, -144.565, 75.677, -189.984]
  Call Extruder(10947.139)
  MoveL 1076 to (-2.97, 13, 50) mm, rotated rx 180 ry 0 rz -180 deg; joints [34.384, 58.836, 14.184, -144.417, 76.053, -189.784]
  Call Extruder(10951.803)
  MoveL 1077 to (-5.78, 12.01, 50) mm, rotated rx 180 ry 0 rz 180 deg; joints [34.5, 58.532, 14.943, -144.364, 76.443, -189.54]
  Call Extruder(10956.466)
  MoveL 1078 to (-8.31, 10.42, 50) mm, rotated rx 180 ry 0 rz -180 deg; joints [34.518, 58.221, 15.723, -144.41, 76.828, -189.263]
  Call Extruder(10961.131)
  MoveL 1079 to (-10.42, 8.31, 50) mm, rotated rx 180 ry 0 rz -180 deg; joints [34.436, 57.92, 16.485, -144.555, 77.19, -188.969]
  Call Extruder(10965.794)
  MoveL 1080 to (-12.01, 5.78, 50) mm, rotated rx 180 ry 0 rz -180 deg; joints [34.254, 57.643, 17.191, -144.795, 77.512, -188.675]
  Call Extruder(10970.458)
  MoveL 1081 to (-13, 2.97, 50) mm, rotated rx 180 ry 0 rz 180 deg; joints [33.981, 57.403, 17.805, -145.118, 77.778, -188.395]
  Call Extruder(10975.122)
  MoveL 1082 to (-13.33, 0, 50) mm, rotated rx 180 ry 0 rz -180 deg; joints [33.63, 57.213, 18.297, -145.511, 77.975, -188.145]
  Call Extruder(10979.786)
  MoveL 1083 to (-13, -2.97, 50) mm, rotated rx 180 ry 0 rz 180 deg; joints [33.218, 57.079, 18.641, -145.953, 78.092, -187.937]
  Call Extruder(10984.449)
  MoveL 1084 to (-12.01, -5.78, 50) mm, rotated rx 180 ry 0 rz -180 deg; joints [32.767, 57.01, 18.821, -146.422, 78.122, -187.781]
  Call Extruder(10989.113)
  MoveL 1085 to (-10.42, -8.31, 50) mm, rotated rx -180 ry 0 rz -180 deg; joints [32.302, 57.008, 18.826, -146.893, 78.062, -187.682]
  Call Extruder(10993.777)
  MoveL 1086 to (-8.31, -10.42, 50) mm, rotated rx -180 ry 0 rz -180 deg; joints [31.85, 57.074, 18.657, -147.339, 77.914, -187.644]
  Call Extruder(10998.441)
  MoveL 1087 to (-5.78, -12.01, 50) mm, rotated rx 180 ry 0 rz 180 deg; joints [31.435, 57.203, 18.322, -147.736, 77.686, -187.668]
  Call Extruder(11003.104)
  MoveL 1088 to (-2.97, -12.99, 50) mm, rotated rx -180 ry 0 rz -180 deg; joints [31.079, 57.391, 17.838, -148.063, 77.387, -187.751]
  Call Extruder(11007.768)
  MoveL 1089 to (0, -13.33, 50) mm, rotated rx 180 ry 0 rz 180 deg; joints [30.801, 57.628, 17.23, -148.301, 77.034, -187.889]
  Call Extruder(11012.432)
  MoveL 1090 to (2.97, -12.99, 50) mm, rotated rx -180 ry 0 rz -180 deg; joints [30.614, 57.903, 16.528, -148.439, 76.645, -188.076]
  Set speed (130.0 mm/s)
  MoveL 1091 to (2.97, -12.99, 55) mm, rotated rx 180 ry 0 rz 180 deg; joints [30.614, 56.972, 16.961, -148.376, 76.22, -188.344]
  MoveL 1092 to (-26.25, -4.54, 55) mm, rotated rx 180 ry 0 rz -180 deg; joints [34.172, 54.98, 22.059, -145.137, 79.307, -187.365]
  Call Extruder(11014.665)
  Set speed (60.0 mm/s)
  MoveL 1093 to (-26.09, -5.96, 55) mm, rotated rx 180 ry 0 rz -180 deg; joints [33.969, 54.918, 22.223, -145.353, 79.364, -187.269]
  Call Extruder(11024.030)
  MoveL 1094 to (-24.12, -11.61, 55) mm, rotated rx -180 ry 0 rz -180 deg; joints [33.033, 54.78, 22.587, -146.322, 79.435, -186.966]
  Call Extruder(11033.395)
  MoveL 1095 to (-20.93, -16.69, 55) mm, rotated rx 180 ry 0 rz -180 deg; joints [32.066, 54.776, 22.597, -147.3, 79.324, -186.782]
  Call Extruder(11042.760)
  MoveL 1096 to (-16.69, -20.93, 55) mm, rotated rx 180 ry 0 rz -180 deg; joints [31.126, 54.906, 22.254, -148.228, 79.034, -186.719]
  Call Extruder(11052.125)
  MoveL 1097 to (-11.61, -24.12, 55) mm, rotated rx -180 ry 0 rz 180 deg; joints [30.272, 55.165, 21.576, -149.05, 78.575, -186.774]
  Call Extruder(11061.489)
  MoveL 1098 to (-5.96, -26.09, 55) mm, rotated rx 180 ry 0 rz 180 deg; joints [29.552, 55.541, 20.599, -149.716, 77.972, -186.938]
  Call Extruder(11070.855)
  MoveL 1099 to (0, -26.77, 55) mm, rotated rx 180 ry 0 rz 180 deg; joints [29.003, 56.018, 19.373, -150.191, 77.256, -187.203]
  Call Extruder(11071.929)
  MoveL 1100 to (0.68, -26.69, 55) mm, rotated rx -180 ry 0 rz -180 deg; joints [28.962, 56.081, 19.212, -150.222, 77.166, -187.244]
  Call Extruder(11080.220)
  MoveL 1101 to (5.96, -26.09, 55) mm, rotated rx 180 ry 0 rz 180 deg; joints [28.65, 56.574, 17.96, -150.452, 76.467, -187.557]
  Call Extruder(11089.585)
  MoveL 1102 to (11.61, -24.11, 55) mm, rotated rx 180 ry 0 rz -180 deg; joints [28.503, 57.184, 16.433, -150.49, 75.648, -187.986]
  Call Extruder(11098.949)
  MoveL 1103 to (16.69, -20.93, 55) mm, rotated rx -180 ry 0 rz 180 deg; joints [28.559, 57.817, 14.866, -150.311, 74.844, -188.478]
  Call Extruder(11108.315)
  MoveL 1104 to (20.93, -16.69, 55) mm, rotated rx -180 ry 0 rz 180 deg; joints [28.808, 58.443, 13.337, -149.931, 74.099, -189.013]
  Call Extruder(11117.680)
  MoveL 1105 to (24.12, -11.61, 55) mm, rotated rx 180 ry 0 rz -180 deg; joints [29.229, 59.028, 11.923, -149.376, 73.451, -189.57]
  Call Extruder(11127.044)
  MoveL 1106 to (26.09, -5.96, 55) mm, rotated rx -180 ry 0 rz 180 deg; joints [29.796, 59.542, 10.692, -148.681, 72.934, -190.125]
  Call Extruder(11136.409)
  MoveL 1107 to (26.77, 0, 55) mm, rotated rx 180 ry 0 rz -180 deg; joints [30.482, 59.956, 9.707, -147.882, 72.572, -190.648]
  Call Extruder(11145.775)
  MoveL 1108 to (26.09, 5.96, 55) mm, rotated rx 180 ry 0 rz -180 deg; joints [31.252, 60.248, 9.017, -147.02, 72.382, -191.112]
  Call Extruder(11155.139)
  MoveL 1109 to (24.11, 11.61, 55) mm, rotated rx 180 ry 0 rz 180 deg; joints [32.076, 60.4, 8.658, -146.137, 72.37, -191.488]
  Call Extruder(11164.504)
  MoveL 1110 to (20.93, 16.69, 55) mm, rotated rx 180 ry 0 rz 180 deg; joints [32.917, 60.405, 8.647, -145.271, 72.535, -191.752]
  Call Extruder(11173.869)
  MoveL 1111 to (16.69, 20.93, 55) mm, rotated rx -180 ry 0 rz -180 deg; joints [33.742, 60.261, 8.986, -144.46, 72.864, -191.886]
  Call Extruder(11183.234)
  MoveL 1112 to (11.61, 24.12, 55) mm, rotated rx 180 ry 0 rz -180 deg; joints [34.517, 59.977, 9.658, -143.737, 73.337, -191.879]
  Call Extruder(11192.599)
  MoveL 1113 to (5.96, 26.09, 55) mm, rotated rx 180 ry 0 rz 180 deg; joints [35.208, 59.569, 10.627, -143.13, 73.929, -191.729]
  Call Extruder(11201.964)
  MoveL 1114 to (0, 26.77, 55) mm, rotated rx 180 ry 0 rz 180 deg; joints [35.784, 59.06, 11.844, -142.665, 74.61, -191.444]
  Call Extruder(11211.329)
  MoveL 1115 to (-5.96, 26.09, 55) mm, rotated rx 180 ry 0 rz -180 deg; joints [36.214, 58.478, 13.25, -142.363, 75.348, -191.038]
  Call Extruder(11220.694)
  MoveL 1116 to (-11.61, 24.12, 55) mm, rotated rx 180 ry 0 rz 180 deg; joints [36.473, 57.854, 14.774, -142.24, 76.108, -190.535]
  Call Extruder(11230.059)
  MoveL 1117 to (-16.69, 20.93, 55) mm, rotated rx -180 ry 0 rz -180 deg; joints [36.542, 57.221, 16.341, -142.308, 76.858, -189.964]
  Call Extruder(11239.424)
  MoveL 1118 to (-20.93, 16.69, 55) mm, rotated rx 180 ry 0 rz 180 deg; joints [36.407, 56.609, 17.873, -142.572, 77.565, -189.358]
  Call Extruder(11248.789)
  MoveL 1119 to (-24.12, 11.61, 55) mm, rotated rx 180 ry 0 rz 180 deg; joints [36.065, 56.048, 19.294, -143.028, 78.197, -188.753]
  Call Extruder(11258.154)
  MoveL 1120 to (-26.09, 5.96, 55) mm, rotated rx 180 ry 0 rz -180 deg; joints [35.528, 55.566, 20.533, -143.663, 78.725, -188.184]
  Call Extruder(11267.519)
  MoveL 1121 to (-26.77, 0, 55) mm, rotated rx 180 ry 0 rz 180 deg; joints [34.817, 55.184, 21.527, -144.451, 79.122, -187.68]
  Call Extruder(11272.308)
  MoveL 1122 to (-26.42, -3.05, 55) mm, rotated rx -180 ry 0 rz -180 deg; joints [34.385, 55.047, 21.886, -144.911, 79.246, -187.468]
  Set speed (130.0 mm/s)
  MoveL 1123 to (-41.86, -6.3, 55) mm, rotated rx -180 ry 0 rz 180 deg; joints [35.393, 53.721, 25.432, -144.118, 81.175, -186.333]
  Call Extruder(11277.306)
  Set speed (60.0 mm/s)
  MoveL 1124 to (-41.51, -9.47, 55) mm, rotated rx 180 ry 0 rz 180 deg; joints [34.924, 53.586, 25.801, -144.611, 81.315, -186.123]
  Call Extruder(11292.201)
  MoveL 1125 to (-38.36, -18.47, 55) mm, rotated rx 180 ry 0 rz -180 deg; joints [33.373, 53.374, 26.386, -146.203, 81.463, -185.675]
  Call Extruder(11307.097)
  MoveL 1126 to (-33.29, -26.54, 55) mm, rotated rx 180 ry 0 rz 180 deg; joints [31.763, 53.368, 26.403, -147.825, 81.316, -185.426]
  Call Extruder(11321.993)
  MoveL 1127 to (-26.54, -33.28, 55) mm, rotated rx 180 ry 0 rz -180 deg; joints [30.206, 53.568, 25.851, -149.365, 80.869, -185.369]
  Call Extruder(11336.889)
  MoveL 1128 to (-18.47, -38.36, 55) mm, rotated rx -180 ry 0 rz -180 deg; joints [28.808, 53.967, 24.761, -150.719, 80.138, -185.486]
  Call Extruder(11351.785)
  MoveL 1129 to (-9.47, -41.5, 55) mm, rotated rx 180 ry 0 rz 180 deg; joints [27.654, 54.552, 23.193, -151.799, 79.163, -185.757]
  Call Extruder(11366.680)
  MoveL 1130 to (0, -42.57, 55) mm, rotated rx 180 ry 0 rz 180 deg; joints [26.805, 55.297, 21.232, -152.547, 77.999, -186.165]
  Call Extruder(11370.520)
  MoveL 1131 to (2.44, -42.3, 55) mm, rotated rx 180 ry 0 rz -180 deg; joints [26.67, 55.519, 20.656, -152.649, 77.67, -186.303]
  Call Extruder(11381.576)
  MoveL 1132 to (9.47, -41.5, 55) mm, rotated rx 180 ry 0 rz -180 deg; joints [26.29, 56.172, 18.979, -152.929, 76.717, -186.697]
  Call Extruder(11396.472)
  MoveL 1133 to (18.47, -38.36, 55) mm, rotated rx 180 ry 0 rz -180 deg; joints [26.114, 57.138, 16.547, -152.944, 75.39, -187.341]
  Call Extruder(11411.368)
  MoveL 1134 to (26.54, -33.28, 55) mm, rotated rx -180 ry 0 rz 180 deg; joints [26.262, 58.148, 14.055, -152.607, 74.092, -188.084]
  Call Extruder(11426.264)
  MoveL 1135 to (33.28, -26.54, 55) mm, rotated rx 180 ry 0 rz 180 deg; joints [26.703, 59.152, 11.624, -151.955, 72.894, -188.906]
  Call Extruder(11441.159)
  MoveL 1136 to (38.36, -18.47, 55) mm, rotated rx 180 ry 0 rz 180 deg; joints [27.4, 60.097, 9.372, -151.035, 71.859, -189.778]
  Call Extruder(11456.055)
  MoveL 1137 to (41.5, -9.47, 55) mm, rotated rx 180 ry 0 rz -180 deg; joints [28.309, 60.933, 7.409, -149.905, 71.038, -190.665]
  Call Extruder(11470.951)
  MoveL 1138 to (42.57, 0, 55) mm, rotated rx 180 ry 0 rz 180 deg; joints [29.382, 61.61, 5.834, -148.629, 70.473, -191.519]
  Call Extruder(11485.847)
  MoveL 1139 to (41.51, 9.47, 55) mm, rotated rx -180 ry 0 rz 180 deg; joints [30.575, 62.088, 4.729, -147.271, 70.188, -192.289]
  Call Extruder(11500.743)
  MoveL 1140 to (38.36, 18.47, 55) mm, rotated rx 180 ry 0 rz -180 deg; joints [31.839, 62.339, 4.152, -145.895, 70.192, -192.924]
  Call Extruder(11515.638)
  MoveL 1141 to (33.28, 26.54, 55) mm, rotated rx 180 ry 0 rz 180 deg; joints [33.128, 62.346, 4.135, -144.561, 70.477, -193.378]
  Call Extruder(11530.534)
  MoveL 1142 to (26.54, 33.29, 55) mm, rotated rx 180 ry 0 rz -180 deg; joints [34.394, 62.109, 4.68, -143.319, 71.022, -193.617]
  Call Extruder(11545.430)
  MoveL 1143 to (18.47, 38.36, 55) mm, rotated rx 180 ry 0 rz -180 deg; joints [35.592, 61.644, 5.755, -142.215, 71.789, -193.62]
  Call Extruder(11560.326)
  MoveL 1144 to (9.47, 41.51, 55) mm, rotated rx -180 ry 0 rz 180 deg; joints [36.675, 60.977, 7.305, -141.285, 72.735, -193.382]
  Call Extruder(11575.222)
  MoveL 1145 to (0, 42.57, 55) mm, rotated rx 180 ry 0 rz 180 deg; joints [37.594, 60.15, 9.247, -140.561, 73.81, -192.917]
  Call Extruder(11590.117)
  MoveL 1146 to (-9.47, 41.5, 55) mm, rotated rx 180 ry 0 rz -180 deg; joints [38.304, 59.21, 11.486, -140.073, 74.964, -192.25]
  Call Extruder(11605.013)
  MoveL 1147 to (-18.47, 38.36, 55) mm, rotated rx 180 ry 0 rz -180 deg; joints [38.762, 58.208, 13.909, -139.846, 76.147, -191.421]
  Call Extruder(11619.909)
  MoveL 1148 to (-26.54, 33.29, 55) mm, rotated rx 180 ry 0 rz -180 deg; joints [38.928, 57.196, 16.401, -139.903, 77.31, -190.479]
  Call Extruder(11634.805)
  MoveL 1149 to (-33.29, 26.54, 55) mm, rotated rx -180 ry 0 rz 180 deg; joints [38.772, 56.227, 18.839, -140.263, 78.41, -189.482]
  Call Extruder(11649.701)
  MoveL 1150 to (-38.36, 18.47, 55) mm, rotated rx 180 ry 0 rz 180 deg; joints [38.277, 55.345, 21.106, -140.934, 79.403, -188.49]
  Call Extruder(11664.596)
  MoveL 1151 to (-41.51, 9.47, 55) mm, rotated rx 180 ry 0 rz -180 deg; joints [37.447, 54.591, 23.088, -141.907, 80.246, -187.565]
  Call Extruder(11679.492)
  MoveL 1152 to (-42.57, 0, 55) mm, rotated rx 180 ry 0 rz 180 deg; joints [36.31, 53.997, 24.681, -143.151, 80.897, -186.761]
  Call Extruder(11687.046)
  MoveL 1153 to (-42.03, -4.8, 55) mm, rotated rx 180 ry 0 rz 180 deg; joints [35.612, 53.785, 25.257, -143.888, 81.11, -186.433]
  Set speed (130.0 mm/s)
  MoveL 1154 to (-54.1, -7.67, 55) mm, rotated rx -180 ry 0 rz 180 deg; joints [36.421, 52.803, 27.985, -143.223, 82.598, -185.5]
  Call Extruder(11691.119)
  Set speed (30.0 mm/s)
  MoveL 1155 to (-53.59, -12.23, 55) mm, rotated rx 180 ry 0 rz 180 deg; joints [35.732, 52.615, 28.518, -143.941, 82.812, -185.206]
  Call Extruder(11702.049)
  MoveL 1156 to (-49.53, -23.85, 55) mm, rotated rx 180 ry 0 rz 180 deg; joints [33.663, 52.349, 29.283, -146.054, 83.043, -184.662]
  Call Extruder(11712.979)
  MoveL 1157 to (-42.98, -34.27, 55) mm, rotated rx 180 ry 0 rz -180 deg; joints [31.506, 52.341, 29.305, -148.221, 82.884, -184.388]
  Call Extruder(11723.910)
  MoveL 1158 to (-34.27, -42.98, 55) mm, rotated rx -180 ry 0 rz -180 deg; joints [29.427, 52.592, 28.583, -150.28, 82.321, -184.362]
  Call Extruder(11734.840)
  MoveL 1159 to (-23.85, -49.53, 55) mm, rotated rx -180 ry 0 rz 180 deg; joints [27.581, 53.096, 27.16, -152.076, 81.372, -184.546]
  Call Extruder(11745.770)
  MoveL 1160 to (-12.23, -53.59, 55) mm, rotated rx -180 ry 0 rz 180 deg; joints [26.087, 53.835, 25.119, -153.488, 80.092, -184.906]
  Call Extruder(11756.700)
  MoveL 1161 to (0, -54.97, 55) mm, rotated rx 180 ry 0 rz 180 deg; joints [25.019, 54.785, 22.574, -154.438, 78.562, -185.418]
  Call Extruder(11760.115)
  MoveL 1162 to (3.82, -54.54, 55) mm, rotated rx 180 ry 0 rz -180 deg; joints [24.823, 55.128, 21.672, -154.588, 78.039, -185.623]
  Call Extruder(11767.630)
  MoveL 1163 to (12.23, -53.59, 55) mm, rotated rx -180 ry 0 rz -180 deg; joints [24.406, 55.906, 19.658, -154.896, 76.878, -186.071]
  Call Extruder(11778.561)
  MoveL 1164 to (23.85, -49.52, 55) mm, rotated rx 180 ry 0 rz 180 deg; joints [24.239, 57.15, 16.517, -154.865, 75.142, -186.86]
  Call Extruder(11789.491)
  MoveL 1165 to (34.27, -42.98, 55) mm, rotated rx 180 ry 0 rz 180 deg; joints [24.487, 58.458, 13.3, -154.379, 73.449, -187.779]
  Call Extruder(11800.421)
  MoveL 1166 to (42.98, -34.27, 55) mm, rotated rx -180 ry 0 rz -180 deg; joints [25.101, 59.765, 10.161, -153.492, 71.891, -188.812]
  Call Extruder(11811.351)
  MoveL 1167 to (49.52, -23.85, 55) mm, rotated rx 180 ry 0 rz -180 deg; joints [26.025, 61.002, 7.247, -152.269, 70.549, -189.93]
  Call Extruder(11822.281)
  MoveL 1168 to (53.59, -12.23, 55) mm, rotated rx 180 ry 0 rz 180 deg; joints [27.2, 62.1, 4.701, -150.788, 69.491, -191.084]
  Call Extruder(11833.212)
  MoveL 1169 to (54.97, 0, 55) mm, rotated rx -180 ry 0 rz -180 deg; joints [28.57, 62.995, 2.653, -149.132, 68.768, -192.214]
  Call Extruder(11844.142)
  MoveL 1170 to (53.59, 12.23, 55) mm, rotated rx -180 ry 0 rz -180 deg; joints [30.077, 63.63, 1.212, -147.388, 68.415, -193.245]
  Call Extruder(11855.072)
  MoveL 1171 to (49.52, 23.85, 55) mm, rotated rx 180 ry 0 rz -180 deg; joints [31.665, 63.963, 0.459, -145.636, 68.441, -194.105]
  Call Extruder(11866.002)
  MoveL 1172 to (42.98, 34.27, 55) mm, rotated rx 180 ry 0 rz 180 deg; joints [33.282, 63.973, 0.437, -143.952, 68.833, -194.725]
  Call Extruder(11876.932)
  MoveL 1173 to (34.27, 42.98, 55) mm, rotated rx 180 ry 0 rz 180 deg; joints [34.874, 63.658, 1.148, -142.396, 69.559, -195.055]
  Call Extruder(11887.863)
  MoveL 1174 to (23.85, 49.53, 55) mm, rotated rx 180 ry 0 rz -180 deg; joints [36.387, 63.04, 2.55, -141.019, 70.568, -195.068]
  Call Extruder(11898.793)
  MoveL 1175 to (12.23, 53.59, 55) mm, rotated rx 180 ry 0 rz -180 deg; joints [37.766, 62.159, 4.565, -139.857, 71.797, -194.759]
  Call Extruder(11909.723)
  MoveL 1176 to (0, 54.97, 55) mm, rotated rx -180 ry 0 rz 180 deg; joints [38.954, 61.071, 7.085, -138.944, 73.181, -194.145]
  Call Extruder(11920.653)
  MoveL 1177 to (-12.23, 53.59, 55) mm, rotated rx 180 ry 0 rz 180 deg; joints [39.895, 59.84, 9.982, -138.31, 74.654, -193.263]
  Call Extruder(11931.583)
  MoveL 1178 to (-23.85, 49.53, 55) mm, rotated rx 180 ry 0 rz 180 deg; joints [40.528, 58.535, 13.112, -137.989, 76.153, -192.165]
  Call Extruder(11942.514)
  MoveL 1179 to (-34.27, 42.98, 55) mm, rotated rx 180 ry 0 rz -180 deg; joints [40.799, 57.226, 16.328, -138.014, 77.624, -190.917]
  Call Extruder(11953.444)
  MoveL 1180 to (-42.98, 34.27, 55) mm, rotated rx 180 ry 0 rz -180 deg; joints [40.659, 55.976, 19.478, -138.417, 79.017, -189.595]
  Call Extruder(11964.374)
  MoveL 1181 to (-49.53, 23.85, 55) mm, rotated rx 180 ry 0 rz 180 deg; joints [40.072, 54.847, 22.412, -139.223, 80.283, -188.282]
  Call Extruder(11975.304)
  MoveL 1182 to (-53.59, 12.23, 55) mm, rotated rx 180 ry 0 rz 180 deg; joints [39.031, 53.886, 24.982, -140.436, 81.374, -187.064]
  Call Extruder(11986.234)
  MoveL 1183 to (-54.97, 0, 55) mm, rotated rx 180 ry 0 rz -180 deg; joints [37.56, 53.133, 27.056, -142.031, 82.237, -186.018]
  Call Extruder(11991.760)
  MoveL 1184 to (-54.27, -6.18, 55) mm, rotated rx -180 ry 0 rz -180 deg; joints [36.644, 52.866, 27.807, -142.99, 82.528, -185.599]
  Set speed (130.0 mm/s)
  MoveL 1185 to (-49.9, -9.51, 55) mm, rotated rx -180 ry 0 rz 180 deg; joints [35.741, 52.997, 27.437, -143.877, 82.248, -185.622]
  MoveL 1186 to (2.97, -12.99, 55) mm, rotated rx 180 ry 0 rz 180 deg; joints [30.614, 56.972, 16.961, -148.376, 76.22, -188.344]
  Call Extruder(11996.424)
  Set speed (80.0 mm/s)
  MoveL 1187 to (5.78, -12.01, 55) mm, rotated rx 180 ry 0 rz -180 deg; joints [30.526, 57.277, 16.201, -148.406, 75.82, -188.568]
  Call Extruder(12001.087)
  MoveL 1188 to (8.31, -10.42, 55) mm, rotated rx 180 ry 0 rz 180 deg; joints [30.538, 57.592, 15.42, -148.331, 75.425, -188.823]
  Call Extruder(12005.751)
  MoveL 1189 to (10.42, -8.31, 55) mm, rotated rx 180 ry 0 rz 180 deg; joints [30.649, 57.901, 14.659, -148.155, 75.058, -189.098]
  Call Extruder(12010.415)
  MoveL 1190 to (12.01, -5.78, 55) mm, rotated rx -180 ry 0 rz -180 deg; joints [30.85, 58.189, 13.954, -147.89, 74.737, -189.38]
  Call Extruder(12015.079)
  MoveL 1191 to (12.99, -2.97, 55) mm, rotated rx 180 ry 0 rz -180 deg; joints [31.131, 58.441, 13.342, -147.55, 74.478, -189.657]
  Call Extruder(12019.743)
  MoveL 1192 to (13.33, 0, 55) mm, rotated rx -180 ry 0 rz -180 deg; joints [31.476, 58.643, 12.852, -147.154, 74.294, -189.913]
  Call Extruder(12024.407)
  MoveL 1193 to (12.99, 2.97, 55) mm, rotated rx 180 ry 0 rz 180 deg; joints [31.869, 58.785, 12.509, -146.72, 74.194, -190.136]
  Call Extruder(12029.070)
  MoveL 1194 to (12.01, 5.78, 55) mm, rotated rx 180 ry 0 rz 180 deg; joints [32.292, 58.859, 12.33, -146.272, 74.182, -190.314]
  Call Extruder(12033.734)
  MoveL 1195 to (10.42, 8.31, 55) mm, rotated rx -180 ry 0 rz 180 deg; joints [32.725, 58.861, 12.325, -145.828, 74.258, -190.436]
  Call Extruder(12038.398)
  MoveL 1196 to (8.31, 10.42, 55) mm, rotated rx 180 ry 0 rz 180 deg; joints [33.149, 58.791, 12.494, -145.411, 74.416, -190.495]
  Call Extruder(12043.062)
  MoveL 1197 to (5.78, 12.01, 55) mm, rotated rx 180 ry 0 rz -180 deg; joints [33.544, 58.653, 12.827, -145.038, 74.649, -190.487]
  Call Extruder(12047.725)
  MoveL 1198 to (2.97, 13, 55) mm, rotated rx 180 ry 0 rz -180 deg; joints [33.893, 58.454, 13.309, -144.727, 74.944, -190.411]
  Call Extruder(12052.389)
  MoveL 1199 to (0, 13.33, 55) mm, rotated rx 180 ry 0 rz 180 deg; joints [34.177, 58.205, 13.915, -144.493, 75.286, -190.272]
  Call Extruder(12057.053)
  MoveL 1200 to (-2.97, 12.99, 55) mm, rotated rx -180 ry 0 rz 180 deg; joints [34.384, 57.919, 14.615, -144.346, 75.659, -190.075]
  Call Extruder(12061.717)
  MoveL 1201 to (-5.78, 12.01, 55) mm, rotated rx 180 ry 0 rz 180 deg; joints [34.5, 57.611, 15.375, -144.294, 76.045, -189.833]
  Call Extruder(12066.380)
  MoveL 1202 to (-8.31, 10.42, 55) mm, rotated rx 180 ry 0 rz -180 deg; joints [34.518, 57.295, 16.155, -144.341, 76.426, -189.558]
  Call Extruder(12071.044)
  MoveL 1203 to (-10.42, 8.31, 55) mm, rotated rx 180 ry 0 rz -180 deg; joints [34.436, 56.989, 16.917, -144.488, 76.784, -189.266]
  Call Extruder(12075.708)
  MoveL 1204 to (-12.01, 5.78, 55) mm, rotated rx -180 ry 0 rz -180 deg; joints [34.254, 56.708, 17.624, -144.729, 77.101, -188.972]
  Call Extruder(12080.372)
  MoveL 1205 to (-13, 2.97, 55) mm, rotated rx 180 ry 0 rz 180 deg; joints [33.981, 56.464, 18.239, -145.054, 77.363, -188.692]
  Call Extruder(12085.036)
  MoveL 1206 to (-13.33, 0, 55) mm, rotated rx -180 ry 0 rz -180 deg; joints [33.63, 56.27, 18.731, -145.448, 77.555, -188.441]
  Call Extruder(12089.700)
  MoveL 1207 to (-13, -2.97, 55) mm, rotated rx -180 ry 0 rz -180 deg; joints [33.218, 56.134, 19.076, -145.892, 77.668, -188.23]
  Call Extruder(12094.363)
  MoveL 1208 to (-12.01, -5.78, 55) mm, rotated rx 180 ry 0 rz -180 deg; joints [32.767, 56.064, 19.255, -146.362, 77.695, -188.071]
  Call Extruder(12099.027)
  MoveL 1209 to (-10.42, -8.31, 55) mm, rotated rx -180 ry 0 rz -180 deg; joints [32.302, 56.062, 19.26, -146.833, 77.633, -187.968]
  Call Extruder(12103.691)
  MoveL 1210 to (-8.31, -10.42, 55) mm, rotated rx 180 ry 0 rz -180 deg; joints [31.85, 56.128, 19.091, -147.279, 77.484, -187.927]
  Call Extruder(12108.355)
  MoveL 1211 to (-5.78, -12.01, 55) mm, rotated rx -180 ry 0 rz -180 deg; joints [31.435, 56.26, 18.755, -147.676, 77.255, -187.947]
  Call Extruder(12113.018)
  MoveL 1212 to (-2.97, -12.99, 55) mm, rotated rx 180 ry 0 rz -180 deg; joints [31.079, 56.451, 18.271, -148.002, 76.957, -188.026]
  Call Extruder(12117.682)
  MoveL 1213 to (0, -13.33, 55) mm, rotated rx -180 ry 0 rz -180 deg; joints [30.801, 56.692, 17.663, -148.239, 76.606, -188.161]
  Call Extruder(12122.346)
  MoveL 1214 to (2.97, -12.99, 55) mm, rotated rx 180 ry 0 rz 180 deg; joints [30.614, 56.972, 16.961, -148.376, 76.22, -188.344]
  Set speed (130.0 mm/s)
  MoveL 1215 to (2.97, -12.99, 60) mm, rotated rx 180 ry 0 rz 180 deg; joints [30.614, 56.045, 17.377, -148.309, 75.785, -188.621]
  MoveL 1216 to (-26.25, -4.54, 60) mm, rotated rx 180 ry 0 rz 180 deg; joints [34.172, 54.017, 22.479, -145.077, 78.861, -187.682]
  Call Extruder(12124.579)
  Set speed (60.0 mm/s)
  MoveL 1217 to (-26.09, -5.96, 60) mm, rotated rx -180 ry 0 rz -180 deg; joints [33.969, 53.953, 22.644, -145.294, 78.916, -187.584]
  Call Extruder(12133.943)
  MoveL 1218 to (-24.12, -11.61, 60) mm, rotated rx 180 ry 0 rz 180 deg; joints [33.033, 53.812, 23.007, -146.264, 78.98, -187.275]
  Call Extruder(12143.308)
  MoveL 1219 to (-20.93, -16.69, 60) mm, rotated rx 180 ry 0 rz 180 deg; joints [32.066, 53.808, 23.018, -147.243, 78.864, -187.084]
  Call Extruder(12152.674)
  MoveL 1220 to (-16.69, -20.93, 60) mm, rotated rx 180 ry 0 rz 180 deg; joints [31.126, 53.941, 22.675, -148.171, 78.571, -187.012]
  Call Extruder(12162.038)
  MoveL 1221 to (-11.61, -24.12, 60) mm, rotated rx 180 ry 0 rz 180 deg; joints [30.272, 54.205, 21.996, -148.992, 78.112, -187.058]
  Call Extruder(12171.403)
  MoveL 1222 to (-5.96, -26.09, 60) mm, rotated rx 180 ry 0 rz 180 deg; joints [29.552, 54.588, 21.017, -149.658, 77.511, -187.214]
  Call Extruder(12180.768)
  MoveL 1223 to (0, -26.77, 60) mm, rotated rx 180 ry 0 rz -180 deg; joints [29.003, 55.074, 19.79, -150.131, 76.799, -187.472]
  Call Extruder(12182.498)
  MoveL 1224 to (1.1, -26.64, 60) mm, rotated rx 180 ry 0 rz 180 deg; joints [28.937, 55.177, 19.531, -150.18, 76.655, -187.536]
  Call Extruder(12190.133)
  MoveL 1225 to (5.96, -26.09, 60) mm, rotated rx 180 ry 0 rz -180 deg; joints [28.65, 55.64, 18.377, -150.389, 76.017, -187.82]
  Call Extruder(12199.498)
  MoveL 1226 to (11.61, -24.11, 60) mm, rotated rx 180 ry 0 rz -180 deg; joints [28.503, 56.26, 16.848, -150.425, 75.206, -188.245]
  Call Extruder(12208.863)
  MoveL 1227 to (16.69, -20.93, 60) mm, rotated rx 180 ry 0 rz -180 deg; joints [28.559, 56.903, 15.281, -150.243, 74.411, -188.734]
  Call Extruder(12218.228)
  MoveL 1228 to (20.93, -16.69, 60) mm, rotated rx 180 ry 0 rz -180 deg; joints [28.808, 57.538, 13.752, -149.86, 73.675, -189.269]
  Call Extruder(12227.593)
  MoveL 1229 to (24.12, -11.61, 60) mm, rotated rx -180 ry 0 rz 180 deg; joints [29.229, 58.131, 12.337, -149.302, 73.037, -189.827]
  Call Extruder(12236.958)
  MoveL 1230 to (26.09, -5.96, 60) mm, rotated rx 180 ry 0 rz 180 deg; joints [29.796, 58.652, 11.107, -148.604, 72.528, -190.384]
  Call Extruder(12246.323)
  MoveL 1231 to (26.77, 0, 60) mm, rotated rx 180 ry 0 rz -180 deg; joints [30.482, 59.071, 10.122, -147.802, 72.174, -190.91]
  Call Extruder(12255.688)
  MoveL 1232 to (26.09, 5.96, 60) mm, rotated rx 180 ry 0 rz -180 deg; joints [31.252, 59.366, 9.433, -146.939, 71.991, -191.379]
  Call Extruder(12265.053)
  MoveL 1233 to (24.11, 11.61, 60) mm, rotated rx 180 ry 0 rz -180 deg; joints [32.076, 59.52, 9.073, -146.054, 71.985, -191.76]
  Call Extruder(12274.418)
  MoveL 1234 to (20.93, 16.69, 60) mm, rotated rx 180 ry 0 rz -180 deg; joints [32.917, 59.525, 9.063, -145.187, 72.154, -192.03]
  Call Extruder(12283.783)
  MoveL 1235 to (16.69, 20.93, 60) mm, rotated rx 180 ry 0 rz -180 deg; joints [33.742, 59.379, 9.402, -144.376, 72.485, -192.17]
  Call Extruder(12293.148)
  MoveL 1236 to (11.61, 24.12, 60) mm, rotated rx 180 ry 0 rz 180 deg; joints [34.517, 59.092, 10.073, -143.653, 72.959, -192.169]
  Call Extruder(12302.513)
  MoveL 1237 to (5.96, 26.09, 60) mm, rotated rx 180 ry 0 rz -180 deg; joints [35.208, 58.679, 11.042, -143.047, 73.55, -192.026]
  Call Extruder(12311.878)
  MoveL 1238 to (0, 26.77, 60) mm, rotated rx -180 ry 0 rz 180 deg; joints [35.784, 58.164, 12.259, -142.583, 74.228, -191.747]
  Call Extruder(12321.243)
  MoveL 1239 to (-5.96, 26.09, 60) mm, rotated rx 180 ry 0 rz -180 deg; joints [36.214, 57.574, 13.665, -142.283, 74.961, -191.347]
  Call Extruder(12330.608)
  MoveL 1240 to (-11.61, 24.12, 60) mm, rotated rx 180 ry 0 rz -180 deg; joints [36.473, 56.941, 15.189, -142.163, 75.715, -190.849]
  Call Extruder(12339.973)
  MoveL 1241 to (-16.69, 20.93, 60) mm, rotated rx 180 ry 0 rz -180 deg; joints [36.542, 56.298, 16.756, -142.234, 76.457, -190.283]
  Call Extruder(12349.338)
  MoveL 1242 to (-20.93, 16.69, 60) mm, rotated rx 180 ry 0 rz 180 deg; joints [36.407, 55.676, 18.289, -142.501, 77.155, -189.68]
  Call Extruder(12358.703)
  MoveL 1243 to (-24.12, 11.61, 60) mm, rotated rx 180 ry 0 rz -180 deg; joints [36.065, 55.105, 19.711, -142.961, 77.777, -189.077]
  Call Extruder(12368.068)
  MoveL 1244 to (-26.09, 5.96, 60) mm, rotated rx -180 ry 0 rz -180 deg; joints [35.528, 54.614, 20.951, -143.599, 78.295, -188.507]
  Call Extruder(12377.433)
  MoveL 1245 to (-26.77, 0, 60) mm, rotated rx -180 ry 0 rz 180 deg; joints [34.817, 54.224, 21.946, -144.389, 78.683, -188.001]
  Call Extruder(12382.222)
  MoveL 1246 to (-26.42, -3.05, 60) mm, rotated rx 180 ry 0 rz 180 deg; joints [34.385, 54.084, 22.306, -144.851, 78.802, -187.786]
  Set speed (130.0 mm/s)
  MoveL 1247 to (-41.86, -6.29, 60) mm, rotated rx -180 ry 0 rz -180 deg; joints [35.393, 52.729, 25.857, -144.065, 80.716, -186.669]
  Call Extruder(12387.219)
  Set speed (60.0 mm/s)
  MoveL 1248 to (-41.51, -9.47, 60) mm, rotated rx 180 ry 0 rz 180 deg; joints [34.924, 52.591, 26.227, -144.559, 80.851, -186.457]
  Call Extruder(12402.115)
  MoveL 1249 to (-38.36, -18.47, 60) mm, rotated rx -180 ry 0 rz 180 deg; joints [33.373, 52.374, 26.813, -146.154, 80.986, -185.998]
  Call Extruder(12417.011)
  MoveL 1250 to (-33.28, -26.54, 60) mm, rotated rx 180 ry 0 rz 180 deg; joints [31.763, 52.367, 26.83, -147.777, 80.83, -185.736]
  Call Extruder(12431.907)
  MoveL 1251 to (-26.54, -33.28, 60) mm, rotated rx 180 ry 0 rz -180 deg; joints [30.206, 52.572, 26.277, -149.317, 80.379, -185.664]
  Call Extruder(12446.803)
  MoveL 1252 to (-18.47, -38.36, 60) mm, rotated rx 180 ry 0 rz 180 deg; joints [28.808, 52.981, 25.185, -150.67, 79.648, -185.765]
  Call Extruder(12461.698)
  MoveL 1253 to (-9.47, -41.5, 60) mm, rotated rx 180 ry 0 rz -180 deg; joints [27.654, 53.579, 23.614, -151.748, 78.677, -186.023]
  Call Extruder(12476.594)
  MoveL 1254 to (0, -42.57, 60) mm, rotated rx -180 ry 0 rz 180 deg; joints [26.805, 54.34, 21.651, -152.493, 77.522, -186.42]
  Call Extruder(12481.090)
  MoveL 1255 to (2.86, -42.25, 60) mm, rotated rx 180 ry 0 rz -180 deg; joints [26.647, 54.605, 20.976, -152.611, 77.14, -186.578]
  Call Extruder(12491.490)
  MoveL 1256 to (9.47, -41.5, 60) mm, rotated rx 180 ry 0 rz 180 deg; joints [26.29, 55.231, 19.396, -152.872, 76.25, -186.943]
  Call Extruder(12506.386)
  MoveL 1257 to (18.47, -38.36, 60) mm, rotated rx 180 ry 0 rz -180 deg; joints [26.114, 56.213, 16.962, -152.882, 74.937, -187.581]
  Call Extruder(12521.282)
  MoveL 1258 to (26.54, -33.28, 60) mm, rotated rx 180 ry 0 rz 180 deg; joints [26.262, 57.239, 14.47, -152.541, 73.653, -188.321]
  Call Extruder(12536.177)
  MoveL 1259 to (33.28, -26.54, 60) mm, rotated rx 180 ry 0 rz -180 deg; joints [26.703, 58.257, 12.039, -151.884, 72.47, -189.142]
  Call Extruder(12551.073)
  MoveL 1260 to (38.36, -18.47, 60) mm, rotated rx 180 ry 0 rz -180 deg; joints [27.4, 59.214, 9.787, -150.96, 71.449, -190.017]
  Call Extruder(12565.969)
  MoveL 1261 to (41.51, -9.47, 60) mm, rotated rx 180 ry 0 rz -180 deg; joints [28.309, 60.059, 7.825, -149.826, 70.643, -190.908]
  Call Extruder(12580.865)
  MoveL 1262 to (42.57, 0, 60) mm, rotated rx 180 ry 0 rz 180 deg; joints [29.382, 60.743, 6.252, -148.545, 70.09, -191.768]
  Call Extruder(12595.761)
  MoveL 1263 to (41.51, 9.47, 60) mm, rotated rx 180 ry 0 rz -180 deg; joints [30.575, 61.226, 5.148, -147.184, 69.815, -192.544]
  Call Extruder(12610.656)
  MoveL 1264 to (38.36, 18.47, 60) mm, rotated rx 180 ry 0 rz 180 deg; joints [31.839, 61.479, 4.572, -145.805, 69.828, -193.187]
  Call Extruder(12625.552)
  MoveL 1265 to (33.28, 26.54, 60) mm, rotated rx 180 ry 0 rz -180 deg; joints [33.128, 61.487, 4.555, -144.469, 70.119, -193.65]
  Call Extruder(12640.448)
  MoveL 1266 to (26.54, 33.29, 60) mm, rotated rx 180 ry 0 rz -180 deg; joints [34.394, 61.248, 5.099, -143.227, 70.667, -193.897]
  Call Extruder(12655.344)
  MoveL 1267 to (18.47, 38.36, 60) mm, rotated rx -180 ry 0 rz -180 deg; joints [35.592, 60.777, 6.173, -142.123, 71.435, -193.909]
